	    //Send message when is new parcel
	    #sx_NewData := (#is_ObjectID <> #ss_Old_Object_ID) AND NOT (#is_ObjectID = '0');
	    // Save last value
	    #ss_Old_Object_ID := #is_ObjectID;

	END_REGION

	REGION 3 – Message array size validation

	    // Get size of the array.
	    #si_MaximumMessageLength := "FC_GetNrOfArrayEl"(#s_UDT_MessageArray.Bytes);

	    // Message array size validation.
	    #ss_Status.InvalidMessageArraySize := WORD_TO_INT(#ci_MessageLength) > #si_MaximumMessageLength;

	END_REGION


	REGION 4 – Message preparation

	    // FIFO full check.
	    IF NOT #iq_UDT_FifoHeader.Status.Full
	    THEN
	        // Errors and send pulse check.
	        IF NOT #ss_Status.FIFOError
	            AND NOT #ss_Status.InvalidMessageArraySize
	            AND #sx_NewData
	        THEN

	            REGION 4.1 – Header preparation

	                // Check sequence number. If it is equal or greater than 255 reset it to 1.
	                IF #iqdi_MessageSequenceNumber <= 255
	                THEN
	                    #iqdi_MessageSequenceNumber += 1;
	                ELSE
	                    #iqdi_MessageSequenceNumber := 1;
	                END_IF;

	                // Write parts of the header into structure.
	                #s_UDT_MessageHeader.SOM := #ci_Som;
	                #s_UDT_MessageHeader.SourceNode := INT_TO_BYTE(#ii_SourceNode);
	                #s_UDT_MessageHeader.DestinationNode := INT_TO_BYTE(#ii_DestinationNode);
	                #s_UDT_MessageHeader.SeqNumber := INT_TO_BYTE(#iqdi_MessageSequenceNumber);
	                #s_UDT_MessageHeader.DataLength := #ci_MessageLength;
	                #s_UDT_MessageHeader.NumMsg := 1;

	                //Convert string value to UDINT
	                #tudi_Temp := STRING_TO_UDINT(#is_ObjectID);

	                // Write parts of the body into structure.
	                #ss_MessageBody.MsgID := #ci_MsgID;
	                #ss_MessageBody.MsgLength := #ci_MsgLength;
	                #ss_MessageBody.ObjectID := UDINT_TO_DWORD(#tudi_Temp);
	                #ss_MessageBody.Eom := #ci_Eom;

	            END_REGION

	            REGION 4.2 – Convert message into array of bytes

	                // Initialize the header serialize position and convert header structure into array of bytes.
	                #sdi_SerializePosition := 0;
	                #si_SerializeStatus := Serialize(SRC_VARIABLE := #s_UDT_MessageHeader,
	                                                 DEST_ARRAY => #s_UDT_MessageArray.Bytes,
	                                                 POS := #sdi_SerializePosition);

	                // Initialize the body serialize position and convert header structure into array of bytes
	                #si_SerializeStatus := Serialize(SRC_VARIABLE := #ss_MessageBody,
	                                                 DEST_ARRAY => #s_UDT_MessageArray.Bytes,
	                                                 POS := #sdi_SerializePosition);

	            END_REGION

	            REGION 4.3 – Write message into the FIFO buffer

	                // Mode 'W' - Write FIFO record.
	                "FC_Fifo"(ic_Mode := 'W',
	                          qUDT_Status => #ss_Status.FIFOStatus,
	                          qx_Error => #ss_Status.FIFOError,
	                          qx_Warning => #ss_Status.FIFOWarning,
	                          iqv_Data := #s_UDT_MessageArray,
	                          iqUDT_FifoHeader := #iq_UDT_FifoHeader,
	                          iqv_DataBuffer := #iqs_FifoData);

	            END_REGION

	        END_IF;
	    ELSE
	        // If FIFO is full set FIFO main and FIFO full errors.
	        #ss_Status.FIFOError := TRUE;
	        #ss_Status.FIFOStatus.FifoFull := TRUE;
	    END_IF;

	END_REGION

	REGION 5 - Status

	    // Parametrization collective error output.
	    #qx_Error :=
	    #ss_Status.FIFOError
	    OR #ss_Status.InvalidTimeInterval
	    OR #ss_Status.InvalidMessageArraySize;

	    // Parametrization collective warning output.
	    #qx_Warning := #ss_Status.FIFOWarning;

	END_REGION
END_FUNCTION_BLOCK

FUNCTION_BLOCK "FB_MFC_Sort_SystemStatus"
{ S7_Optimized_Access := 'TRUE' }
VERSION : 0.1
// ATTRIBUTES
// AUTO_NUMBER = True
// BLOCK_NUMBER = 125
// END_ATTRIBUTES
   VAR_INPUT
      ii_SystemStatus { ExternalAccessible := 'False'; ExternalVisible := 'False'; ExternalWritable := 'False'} : Int;   // 1 - System stopped, 2 - System running
      iw_SystemMode { ExternalAccessible := 'False'; ExternalVisible := 'False'; ExternalWritable := 'False'} : Word;   // Bit value according to the documentation
      iui_LocationIdentifier { ExternalAccessible := 'False'; ExternalVisible := 'False'; ExternalWritable := 'False'} : UInt;   // Location Identifier
      ii_SourceNode { ExternalAccessible := 'False'; ExternalVisible := 'False'; ExternalWritable := 'False'} : Int;   // ID Source Node
      ii_DestinationNode { ExternalAccessible := 'False'; ExternalVisible := 'False'; ExternalWritable := 'False'} : Int;   // ID Destination Node
      ix_SendAllStatuses { ExternalAccessible := 'False'; ExternalVisible := 'False'; ExternalWritable := 'False'} : Bool;   // True - update all the statuses
   END_VAR

   VAR_OUTPUT
      qx_Error { ExternalAccessible := 'False'; ExternalVisible := 'False'; ExternalWritable := 'False'} : Bool;   // TRUE when collective block error occurred
      qx_Warning { ExternalAccessible := 'False'; ExternalVisible := 'False'; ExternalWritable := 'False'} : Bool;   // TRUE when collective block warning occurred
   END_VAR

   VAR_IN_OUT
      iq_UDT_FifoHeader : "UDT_FifoHeader";   // FIFO header
      iqs_FifoData : Array[*] of "UDT_MessageV2";   // FIFO data buffer
      iqdi_MessageSequenceNumber { ExternalAccessible := 'False'; ExternalVisible := 'False'; ExternalWritable := 'False'} : Int;   // Message number
   END_VAR

   VAR
      s_UDT_MessageArray { ExternalAccessible := 'False'; ExternalVisible := 'False'; ExternalWritable := 'False'; S7_SetPoint := 'False'} : "UDT_MessageV2";   // Message array byte
      s_UDT_MessageHeader { ExternalAccessible := 'False'; ExternalVisible := 'False'; ExternalWritable := 'False'; S7_SetPoint := 'False'} : "UDT_MFCSortMessageHeader";   // Message header
      s_F_TRIG_SendAllStatuses {InstructionName := 'F_TRIG'; LibVersion := '1.0'; ExternalAccessible := 'False'; ExternalVisible := 'False'; ExternalWritable := 'False'; S7_SetPoint := 'False'} : F_TRIG;   // Falling edge trigger from signal send all statuses
      ss_MessageBody { ExternalAccessible := 'False'; ExternalVisible := 'False'; ExternalWritable := 'False'} : Struct   // Message body
         MsgID { ExternalAccessible := 'False'; ExternalVisible := 'False'; ExternalWritable := 'False'} : Word;   // Message ID
         MsgLength { ExternalAccessible := 'False'; ExternalVisible := 'False'; ExternalWritable := 'False'} : Word;   // Message length
         LocationIdentifier { ExternalAccessible := 'False'; ExternalVisible := 'False'; ExternalWritable := 'False'} : Word;   // Location Identifier
         SystemStatus { ExternalAccessible := 'False'; ExternalVisible := 'False'; ExternalWritable := 'False'} : Byte;   // System status
         SystemMode { ExternalAccessible := 'False'; ExternalVisible := 'False'; ExternalWritable := 'False'} : Word;   // System mode
         Eom { ExternalAccessible := 'False'; ExternalVisible := 'False'; ExternalWritable := 'False'} : Byte;   // End of message
         Test { ExternalAccessible := 'False'; ExternalVisible := 'False'; ExternalWritable := 'False'} : Word := 16#0011;
         Test_1 { ExternalAccessible := 'False'; ExternalVisible := 'False'; ExternalWritable := 'False'} : Byte := 16#22;
      END_STRUCT;
      ss_Status { ExternalAccessible := 'False'; ExternalVisible := 'False'; ExternalWritable := 'False'} : Struct   // Status structure
         FIFOStatus { ExternalAccessible := 'False'; ExternalVisible := 'False'; ExternalWritable := 'False'} : "UDT_FifoStatus";
         FIFOError { ExternalAccessible := 'False'; ExternalVisible := 'False'; ExternalWritable := 'False'; S7_SetPoint := 'True'} : Bool;   //  FIFO error
         FIFOWarning { ExternalAccessible := 'False'; ExternalVisible := 'False'; ExternalWritable := 'False'; S7_SetPoint := 'True'} : Bool;   // FIFO warning
         InvalidMessageArraySize { ExternalAccessible := 'False'; ExternalVisible := 'False'; ExternalWritable := 'False'} : Bool;   // Message array is too short for message
         InvalidTimeInterval { ExternalAccessible := 'False'; ExternalVisible := 'False'; ExternalWritable := 'False'} : Bool;   // Heartbeat time interval lower than zero
      END_STRUCT;
      sw_SystemMode { ExternalAccessible := 'False'; ExternalVisible := 'False'; ExternalWritable := 'False'} : Word := 0;   // Bit value according to the documentation
      sw_Old_SystemMode { ExternalAccessible := 'False'; ExternalVisible := 'False'; ExternalWritable := 'False'} : Word;   // Data from previous PLC cycle: Maximum number of elements in message array
      sdi_SerializePosition { ExternalAccessible := 'False'; ExternalVisible := 'False'; ExternalWritable := 'False'} : DInt;   // Position in array where serialize finished writing data +1
      si_MaximumMessageLength { ExternalAccessible := 'False'; ExternalVisible := 'False'; ExternalWritable := 'False'} : Int;   // Maximum number of elements in message array
      si_SerializeStatus { ExternalAccessible := 'False'; ExternalVisible := 'False'; ExternalWritable := 'False'} : Int;   // Function serialize status
      si_SystemStatus { ExternalAccessible := 'False'; ExternalVisible := 'False'; ExternalWritable := 'False'} : Int := 0;   // 1 - System stopped, 2 - System running
      si_Old_SystemStatus { ExternalAccessible := 'False'; ExternalVisible := 'False'; ExternalWritable := 'False'} : Int := 0;   // Data from previous PLC cycle: 0 - System stopped, 1 - System running
      sx_NewData { ExternalAccessible := 'False'; ExternalVisible := 'False'; ExternalWritable := 'False'} : Bool;   // True - send a message to the MFC
   END_VAR

   VAR CONSTANT
      ci_MessageLength : Word := 16#0009;   // 10#0009 = 16#0009 - Message length
      ci_Som : Byte := 16#FD;   // Start of message
      ci_Eom : Byte := 16#FE;   // End of message
      ci_MsgID : Word := 16#00CC;   // 10#0204 = 16#00CC - Message ID
      ci_MsgLength : Word := 16#0005;   // 10#0005 = 16#0005 - Message length
   END_VAR


BEGIN
	(*
	----------------------------------------------------------------------------------------
	|                                                                                      |
	|  Copyright  2023             FORTNA Europe BV                                        |
	|  All Rights Reserved         Netherlands                                             |
	|                                                                                      |
	----------------------------------------------------------------------------------------
	Version history:
	Date        | Version   | Author       | Remark
	----------------------------------------------------------------------------------------
	21/07/2023  | 1.0       | S. Nikodem   | Release TIA 17 | DHL Munich 2023
	23/08/2023  | 1.1       | S. Theocharis| Serialise byte issue 0 - quick fix
	19/10/2023  | 1.2       | S. Nikodem   | Added "ix_SendAllStatuses" input and update for Serialize structure
	13/03/2023  | 1.3       | S. Nieswiec  | Updated for new Baseline
	02/05/2024  | 1.4       | J.Majer      | Datatype conversions changed from automatic to explicit, to accomodate IEC 61131-3 standard

	*)

	REGION 1 – FIFO header status update

	    // Mode 'S' - FIFO register status update.
	    "FC_Fifo"(ic_Mode := 'S',
	              qUDT_Status => #ss_Status.FIFOStatus,
	              qx_Error => #ss_Status.FIFOError,
	              qx_Warning => #ss_Status.FIFOWarning,
	              iqv_Data := #s_UDT_MessageArray,
	              iqUDT_FifoHeader := #iq_UDT_FifoHeader,
	              iqv_DataBuffer := #iqs_FifoData);

	END_REGION

	REGION 2 – Data preparation

	    // Prepare trigger
	    #s_F_TRIG_SendAllStatuses(CLK := #ix_SendAllStatuses);

	    // Data preparation
	    //  1 - System stopped, 2 - System running
	    #si_SystemStatus := #ii_SystemStatus;
	    // Bit value according to the documentation
	    #sw_SystemMode := #iw_SystemMode;

	    //Check if the data from the previous PLC cycle differs, if so, send a message to the MFC.
	    #sx_NewData := (#si_Old_SystemStatus <> #si_SystemStatus) OR (#sw_Old_SystemMode <> #sw_SystemMode) OR #s_F_TRIG_SendAllStatuses.Q;

	    // Copy data
	    #si_Old_SystemStatus := #si_SystemStatus;
	    #sw_Old_SystemMode := #sw_SystemMode;

	END_REGION

	REGION 3 – Message array size validation

	    // Get size of the array.
	    #si_MaximumMessageLength := "FC_GetNrOfArrayEl"(#s_UDT_MessageArray.Bytes);

	    // Message array size validation.
	    #ss_Status.InvalidMessageArraySize := WORD_TO_INT(#ci_MessageLength) > #si_MaximumMessageLength;

	END_REGION

	REGION 4 – Message preparation

	    // FIFO full check.
	    IF NOT #iq_UDT_FifoHeader.Status.Full
	    THEN
	        // Errors and send pulse check.
	        IF NOT #ss_Status.FIFOError
	            AND NOT #ss_Status.InvalidMessageArraySize
	            AND #sx_NewData
	        THEN

	            REGION 4.1 – Header preparation

	                // Check sequence number. If it is equal or greater than 255 reset it to 1.
	                IF #iqdi_MessageSequenceNumber <= 255
	                THEN
	                    #iqdi_MessageSequenceNumber += 1;
	                ELSE
	                    #iqdi_MessageSequenceNumber := 1;
	                END_IF;

	                // Write parts of the header into structure.
	                // Write parts of the header into structure.
	                #s_UDT_MessageHeader.SOM := #ci_Som;
	                #s_UDT_MessageHeader.SourceNode := INT_TO_BYTE(#ii_SourceNode);
	                #s_UDT_MessageHeader.DestinationNode := INT_TO_BYTE(#ii_DestinationNode);
	                #s_UDT_MessageHeader.SeqNumber := INT_TO_BYTE(#iqdi_MessageSequenceNumber);
	                #s_UDT_MessageHeader.DataLength := #ci_MessageLength;
	                #s_UDT_MessageHeader.NumMsg := 1;

	                // Write parts of the body into structure.
	                #ss_MessageBody.MsgID := #ci_MsgID;
	                #ss_MessageBody.MsgLength := #ci_MsgLength;
	                #ss_MessageBody.LocationIdentifier := DINT_TO_WORD(#iui_LocationIdentifier);
	                #ss_MessageBody.SystemStatus := INT_TO_BYTE(#si_SystemStatus);
	                #ss_MessageBody.SystemMode := #sw_SystemMode;
	                #ss_MessageBody.Eom := #ci_Eom;

	            END_REGION

	            REGION 4.2 – Convert message into array of bytes

	                // Initialize the header serialize position and convert header structure into array of bytes.
	                #sdi_SerializePosition := 0;
	                #si_SerializeStatus := Serialize(SRC_VARIABLE := #s_UDT_MessageHeader,
	                                                 DEST_ARRAY => #s_UDT_MessageArray.Bytes,
	                                                 POS := #sdi_SerializePosition);

	                #si_SerializeStatus := Serialize(SRC_VARIABLE := #ss_MessageBody.MsgID,
	                                                 DEST_ARRAY => #s_UDT_MessageArray.Bytes,
	                                                 POS := #sdi_SerializePosition);

	                #si_SerializeStatus := Serialize(SRC_VARIABLE := #ss_MessageBody.MsgLength,
	                                                 DEST_ARRAY => #s_UDT_MessageArray.Bytes,
	                                                 POS := #sdi_SerializePosition);

	                #si_SerializeStatus := Serialize(SRC_VARIABLE := #ss_MessageBody.LocationIdentifier,
	                                                 DEST_ARRAY => #s_UDT_MessageArray.Bytes,
	                                                 POS := #sdi_SerializePosition);

	                #si_SerializeStatus := Serialize(SRC_VARIABLE := #ss_MessageBody.SystemStatus,
	                                                 DEST_ARRAY => #s_UDT_MessageArray.Bytes,
	                                                 POS := #sdi_SerializePosition);

	                #si_SerializeStatus := Serialize(SRC_VARIABLE := #ss_MessageBody.SystemMode,
	                                                 DEST_ARRAY => #s_UDT_MessageArray.Bytes,
	                                                 POS := #sdi_SerializePosition);

	                #si_SerializeStatus := Serialize(SRC_VARIABLE := #ss_MessageBody.Eom,
	                                                 DEST_ARRAY => #s_UDT_MessageArray.Bytes,
	                                                 POS := #sdi_SerializePosition);

	            END_REGION

	            REGION 4.3 – Write message into the FIFO buffer

	                // Mode 'W' - Write FIFO record.
	                "FC_Fifo"(ic_Mode := 'W',
	                          qUDT_Status => #ss_Status.FIFOStatus,
	                          qx_Error => #ss_Status.FIFOError,
	                          qx_Warning => #ss_Status.FIFOWarning,
	                          iqv_Data := #s_UDT_MessageArray,
	                          iqUDT_FifoHeader := #iq_UDT_FifoHeader,
	                          iqv_DataBuffer := #iqs_FifoData);

	            END_REGION

	        END_IF;
	    ELSE
	        // If FIFO is full set FIFO main and FIFO full errors.
	        #ss_Status.FIFOError := TRUE;
	        #ss_Status.FIFOStatus.FifoFull := TRUE;
	    END_IF;

	END_REGION

	REGION 5 - Status

	    // Parametrization collective error output.
	    #qx_Error :=
	    #ss_Status.FIFOError
	    OR #ss_Status.InvalidTimeInterval
	    OR #ss_Status.InvalidMessageArraySize;

	    // Parametrization collective warning output.
	    #qx_Warning := #ss_Status.FIFOWarning;

	END_REGION
END_FUNCTION_BLOCK

FUNCTION_BLOCK "FB_MFC_Sort_TCPIPSend"
TITLE = FB_TCPIPSend
{ S7_Optimized_Access := 'TRUE' }
AUTHOR : MHSE
FAMILY : Communication
VERSION : 2.0
// ATTRIBUTES
// AUTO_NUMBER = True
// BLOCK_NUMBER = 127
// END_ATTRIBUTES
//Function block to send data from TCPIP.
   VAR_INPUT
      i_UDT_Connection { ExternalAccessible := 'False'; ExternalVisible := 'False'; ExternalWritable := 'False'} : "UDT_Connection";   // Connection parameters
      ix_EnableSend { ExternalAccessible := 'False'; ExternalVisible := 'False'; ExternalWritable := 'False'} : Bool;   // TRUE when send is enable
   END_VAR

   VAR_OUTPUT
      qx_Error { ExternalAccessible := 'False'; ExternalVisible := 'False'; ExternalWritable := 'False'} : Bool;   // TRUE when collective block error occurred
      qx_Warning { ExternalAccessible := 'False'; ExternalVisible := 'False'; ExternalWritable := 'False'} : Bool;   // TRUE when collective block warning occurred
   END_VAR

   VAR_IN_OUT
      iq_UDT_FifoLowHeader : "UDT_FifoHeader";   // Low priority FIFO header
      iqs_FifoLowData : Variant;   // Low priority FIFO data
      iq_UDT_FifoMediumHeader : "UDT_FifoHeader";   // Medium priority FIFO header
      iqs_FifoMediumData : Variant;   // Medium priority FIFO data
      iq_UDT_FifoHighHeader : "UDT_FifoHeader";   // High priority FIFO header
      iqs_FifoHighData : Variant;   // High priority FIFO data
   END_VAR

   VAR
      s_FB_TSEND {InstructionName := 'TSEND'; LibVersion := '4.0'; ExternalAccessible := 'False'; ExternalVisible := 'False'; ExternalWritable := 'False'; S7_SetPoint := 'False'} : TSEND;   // Siemens "TSEND" block - to send the data over TCPIP socket
      s_UDT_MessageArray { ExternalAccessible := 'False'; ExternalVisible := 'False'; ExternalWritable := 'False'; S7_SetPoint := 'False'} : "UDT_MessageV2";   // Message
      ss_TSEND { ExternalAccessible := 'False'; ExternalVisible := 'False'; ExternalWritable := 'False'} : Struct   // TSEND block structure
         Status { ExternalAccessible := 'False'; ExternalVisible := 'False'; ExternalWritable := 'False'} : Word;   //    TSEND - Status
         Request { ExternalAccessible := 'False'; ExternalVisible := 'False'; ExternalWritable := 'False'} : Bool;   //    TSEND - Request
         Busy { ExternalAccessible := 'False'; ExternalVisible := 'False'; ExternalWritable := 'False'} : Bool;   //    TSEND - Busy
         Done { ExternalAccessible := 'False'; ExternalVisible := 'False'; ExternalWritable := 'False'} : Bool;   //    TSEND - Done
         Error { ExternalAccessible := 'False'; ExternalVisible := 'False'; ExternalWritable := 'False'} : Bool;   //    TSEND - Error
      END_STRUCT;
      ss_Status { ExternalAccessible := 'False'; ExternalVisible := 'False'; ExternalWritable := 'False'} : Struct   // Status structure
         FIFOLowPriorityStatus { ExternalAccessible := 'False'; ExternalVisible := 'False'; ExternalWritable := 'False'} : "UDT_FifoStatus";
         FIFOMedPriorityStatus { ExternalAccessible := 'False'; ExternalVisible := 'False'; ExternalWritable := 'False'} : "UDT_FifoStatus";
         FIFOHighPriorityStatus { ExternalAccessible := 'False'; ExternalVisible := 'False'; ExternalWritable := 'False'} : "UDT_FifoStatus";
         FIFOLowPriorityError { ExternalAccessible := 'False'; ExternalVisible := 'False'; ExternalWritable := 'False'} : Bool;   // FIFO low priority error
         FIFOLowPriorityWarning { ExternalAccessible := 'False'; ExternalVisible := 'False'; ExternalWritable := 'False'} : Bool;   // FIFO low priority warning
         FIFOMedPriorityError { ExternalAccessible := 'False'; ExternalVisible := 'False'; ExternalWritable := 'False'} : Bool;   // FIFO medium priority error
         FIFOMedPriorityWarning { ExternalAccessible := 'False'; ExternalVisible := 'False'; ExternalWritable := 'False'} : Bool;   // FIFO medium priority warning
         FIFOHighPriorityError { ExternalAccessible := 'False'; ExternalVisible := 'False'; ExternalWritable := 'False'} : Bool;   // FIFO high priority error
         FIFOHighPriorityWarning { ExternalAccessible := 'False'; ExternalVisible := 'False'; ExternalWritable := 'False'} : Bool;   // FIFO high priority warning
         SendError { ExternalAccessible := 'False'; ExternalVisible := 'False'; ExternalWritable := 'False'} : Bool;   // Send operation error
      END_STRUCT;
      sw_BodyLength { ExternalAccessible := 'False'; ExternalVisible := 'False'; ExternalWritable := 'False'} : Word;   // Message body length
      sa_BodyLength { ExternalAccessible := 'False'; ExternalVisible := 'False'; ExternalWritable := 'False'} : Array[0..1] of Byte;
      si_MessageLength { ExternalAccessible := 'False'; ExternalVisible := 'False'; ExternalWritable := 'False'} : Int;   // Message length
      sx_MessageReady { ExternalAccessible := 'False'; ExternalVisible := 'False'; ExternalWritable := 'False'} : Bool;   // Message is ready to send
      sx_MessageRead { ExternalAccessible := 'False'; ExternalVisible := 'False'; ExternalWritable := 'False'} : Bool;   // Message has been read
      sx_MessageReadRequest { ExternalAccessible := 'False'; ExternalVisible := 'False'; ExternalWritable := 'False'} : Bool;   // Request to read message
      sx_FIFOError { ExternalAccessible := 'False'; ExternalVisible := 'False'; ExternalWritable := 'False'} : Bool;   // Summary FIFO error
      sdi_SerializePosition { ExternalAccessible := 'False'; ExternalVisible := 'False'; ExternalWritable := 'False'} : DInt;   // Position in array where serialize finished writing data +1
      si_SerializeStatus { ExternalAccessible := 'False'; ExternalVisible := 'False'; ExternalWritable := 'False'} : Int;   // Function serialize status
   END_VAR

   VAR CONSTANT
      ci_HeaderLength : Int := 8;   // Message header length
      ci_BodyLengthPosition : Int := 4;   // Position in header where message body length value starts
      cdi_POS : DInt := 2;
   END_VAR


BEGIN
	(*
	----------------------------------------------------------------------------------------
	|                                                                                      |
	|  Copyright  2023             FORTNA Europe BV                                        |
	|  All Rights Reserved         Netherlands                                             |
	|                                                                                      |
	----------------------------------------------------------------------------------------
	Version history:
	Date        | Version   | Author       | Remark
	----------------------------------------------------------------------------------------
	16/01/2023  | 1.0       | S. Nikodem   | Release TIA 17 | DHL Munich 2023
	13/03/2023  | 1.1       | S. Nieswiec  | Updated for new Baseline
	*)

	REGION 1 – Update FIFO header status bits

	    // Mode 'S' - High priority FIFO register status update.
	    "FC_Fifo"(ic_Mode := 'S',
	              qUDT_Status => #ss_Status.FIFOHighPriorityStatus,
	              qx_Error => #ss_Status.FIFOHighPriorityError,
	              qx_Warning => #ss_Status.FIFOHighPriorityWarning,
	              iqv_Data := #s_UDT_MessageArray,
	              iqUDT_FifoHeader := #iq_UDT_FifoHighHeader,
	              iqv_DataBuffer := #iqs_FifoHighData);

	    // Mode 'S' - Medium priority FIFO register status update.
	    "FC_Fifo"(ic_Mode := 'S',
	              qUDT_Status => #ss_Status.FIFOMedPriorityStatus,
	              qx_Error => #ss_Status.FIFOMedPriorityError,
	              qx_Warning => #ss_Status.FIFOMedPriorityWarning,
	              iqv_Data := #s_UDT_MessageArray,
	              iqUDT_FifoHeader := #iq_UDT_FifoMediumHeader,
	              iqv_DataBuffer := #iqs_FifoMediumData);

	    // Mode 'S' - Low priority FIFO register status update.
	    "FC_Fifo"(ic_Mode := 'S',
	              qUDT_Status => #ss_Status.FIFOLowPriorityStatus,
	              qx_Error => #ss_Status.FIFOLowPriorityError,
	              qx_Warning => #ss_Status.FIFOLowPriorityWarning,
	              iqv_Data := #s_UDT_MessageArray,
	              iqUDT_FifoHeader := #iq_UDT_FifoLowHeader,
	              iqv_DataBuffer := #iqs_FifoLowData);

	END_REGION

	REGION 2 – FIFO header summary error

	    #sx_FIFOError :=
	    #ss_Status.FIFOHighPriorityError
	    OR #ss_Status.FIFOMedPriorityError
	    OR #ss_Status.FIFOLowPriorityError;

	END_REGION

	REGION 3 – FIFO Read request

	    #sx_MessageReadRequest :=
	    #ix_EnableSend
	    AND NOT #sx_FIFOError
	    AND NOT #ss_TSEND.Error
	    AND #ss_TSEND.Status = 16#7000;

	END_REGION

	REGION 4 – Read the message from high priority FIFO data buffer

	    IF #sx_MessageReadRequest
	        AND NOT #iq_UDT_FifoHighHeader.Status.Empty
	        AND NOT #sx_MessageRead
	    THEN
	        // Mode 'R' - Read high priority FIFO record.
	        "FC_Fifo"(ic_Mode := 'R',
	                  qUDT_Status => #ss_Status.FIFOHighPriorityStatus,
	                  qx_Error => #ss_Status.FIFOHighPriorityError,
	                  qx_Warning => #ss_Status.FIFOHighPriorityWarning,
	                  iqv_Data := #s_UDT_MessageArray,
	                  iqUDT_FifoHeader := #iq_UDT_FifoHighHeader,
	                  iqv_DataBuffer := #iqs_FifoHighData);

	        #sx_MessageRead := TRUE;
	    END_IF;

	END_REGION

	REGION 5 – Read the message from medium priority FIFO data buffer

	    IF #sx_MessageReadRequest
	        AND #iq_UDT_FifoHighHeader.Status.Empty
	        AND NOT #iq_UDT_FifoMediumHeader.Status.Empty
	        AND NOT #sx_MessageRead
	    THEN
	        // Mode 'R' - Read medium priority FIFO record.
	        "FC_Fifo"(ic_Mode := 'R',
	                  qUDT_Status => #ss_Status.FIFOMedPriorityStatus,
	                  qx_Error => #ss_Status.FIFOMedPriorityError,
	                  qx_Warning => #ss_Status.FIFOMedPriorityWarning,
	                  iqv_Data := #s_UDT_MessageArray,
	                  iqUDT_FifoHeader := #iq_UDT_FifoMediumHeader,
	                  iqv_DataBuffer := #iqs_FifoMediumData);

	        #sx_MessageRead := TRUE;
	    END_IF;

	END_REGION

	REGION 6 – Read the message from low priority FIFO data buffer

	    IF #sx_MessageReadRequest
	        AND #iq_UDT_FifoHighHeader.Status.Empty
	        AND #iq_UDT_FifoMediumHeader.Status.Empty
	        AND NOT #iq_UDT_FifoLowHeader.Status.Empty
	        AND NOT #sx_MessageRead
	    THEN
	        #sx_MessageRead := TRUE;

	        // Mode 'R' - Read low priority FIFO record.
	        "FC_Fifo"(ic_Mode := 'R',
	                  qUDT_Status => #ss_Status.FIFOLowPriorityStatus,
	                  qx_Error => #ss_Status.FIFOLowPriorityError,
	                  qx_Warning => #ss_Status.FIFOLowPriorityWarning,
	                  iqv_Data := #s_UDT_MessageArray,
	                  iqUDT_FifoHeader := #iq_UDT_FifoLowHeader,
	                  iqv_DataBuffer := #iqs_FifoLowData);
	    END_IF;

	END_REGION

	REGION 7 – Message length

	    // Measuring the length of a read message.
	    IF #sx_MessageRead
	        AND NOT #sx_MessageReady
	    THEN
	        // Initialize the message length.
	        #si_MessageLength := 0;

	        // Get the length of the message by extracting the body length from the message header.
	        #sa_BodyLength[0] := #s_UDT_MessageArray.Bytes[#ci_BodyLengthPosition];
	        #sa_BodyLength[1] := #s_UDT_MessageArray.Bytes[#ci_BodyLengthPosition + 1];

	        #sdi_SerializePosition := 0;
	        #si_SerializeStatus := Deserialize(SRC_ARRAY := #sa_BodyLength,
	                                           DEST_VARIABLE => #sw_BodyLength,
	                                           POS := #sdi_SerializePosition);

	        #si_MessageLength := WORD_TO_INT(#sw_BodyLength) + #ci_HeaderLength + 1; // Add body, header and tail
	        #sx_MessageReady := TRUE;
	    END_IF;

	END_REGION

	REGION 8 – Send request

	    IF #sx_MessageRead
	        AND #sx_MessageReady
	    THEN
	        #ss_TSEND.Request := TRUE;
	    END_IF;

	END_REGION

	REGION 9 – Send data

	    #s_FB_TSEND(REQ := #ss_TSEND.Request,
	                ID := #i_UDT_Connection.ID,
	                LEN := INT_TO_UDINT(#si_MessageLength),
	                DONE => #ss_TSEND.Done,
	                BUSY => #ss_TSEND.Busy,
	                ERROR => #ss_TSEND.Error,
	                STATUS => #ss_TSEND.Status,
	                DATA := #s_UDT_MessageArray);

	    // Reset send request, message read and ready bits.
	    IF #ss_TSEND.Request
	        AND NOT #ss_TSEND.Busy
	        AND (#ss_TSEND.Done
	        OR #ss_TSEND.Status = 16#7000)
	    THEN
	        #ss_TSEND.Request := FALSE;
	        #sx_MessageRead := FALSE;
	        #sx_MessageReady := FALSE;
	    END_IF;

	    // Reset send error and TSEND status after correctly sent message.
	    IF #ss_TSEND.Done
	    THEN
	        #ss_Status.SendError := FALSE;
	    END_IF;

	    // Set send error and TSEND status if error occured.
	    IF #ss_TSEND.Error
	    THEN
	        #ss_Status.SendError := TRUE;
	    END_IF;

	END_REGION

	REGION 10 – Status

	    // Parametrization collective error output.
	    #qx_Error :=
	    #sx_FIFOError
	    OR #ss_Status.SendError;

	    // Parametrization collective warning output.
	    #qx_Warning :=
	    #ss_Status.FIFOHighPriorityWarning
	    OR #ss_Status.FIFOMedPriorityWarning
	    OR #ss_Status.FIFOLowPriorityWarning;

	END_REGION
END_FUNCTION_BLOCK

FUNCTION_BLOCK "FB_MFC_Sort_VIDResponse"
{ S7_Optimized_Access := 'TRUE' }
VERSION : 0.1
// ATTRIBUTES
// AUTO_NUMBER = True
// BLOCK_NUMBER = 128
// END_ATTRIBUTES
   VAR_INPUT
      ii_Object_ID { ExternalAccessible := 'False'; ExternalVisible := 'False'; ExternalWritable := 'False'} : Int;   // Parcel identifier
      i_ActualTimeDTL {InstructionName := 'DTL'; LibVersion := '1.0'; ExternalAccessible := 'False'; ExternalVisible := 'False'; ExternalWritable := 'False'} : DTL;   // Actual date and time in DTL
      ii_SourceNode { ExternalAccessible := 'False'; ExternalVisible := 'False'; ExternalWritable := 'False'} : Int;   // ID Source Node
      ii_DestinationNode { ExternalAccessible := 'False'; ExternalVisible := 'False'; ExternalWritable := 'False'} : Int;   // ID Destination Node
   END_VAR

   VAR_OUTPUT
      qx_Error { ExternalAccessible := 'False'; ExternalVisible := 'False'; ExternalWritable := 'False'} : Bool;   // TRUE when collective block error occurred
      qx_Warning { ExternalAccessible := 'False'; ExternalVisible := 'False'; ExternalWritable := 'False'} : Bool;   // TRUE when collective block warning occurred
   END_VAR

   VAR_IN_OUT
      iq_UDT_FifoHeader : "UDT_FifoHeader";   // FIFO header
      iqs_FifoData : Array[*] of "UDT_MessageV2";   // FIFO data buffer
      iqdi_MessageSequenceNumber { ExternalAccessible := 'False'; ExternalVisible := 'False'; ExternalWritable := 'False'} : Int;   // Message number
   END_VAR

   VAR
      s_UDT_MessageArray { ExternalAccessible := 'False'; ExternalVisible := 'False'; ExternalWritable := 'False'; S7_SetPoint := 'False'} : "UDT_MessageV2";   // Message array byte
      s_UDT_MessageHeader { ExternalAccessible := 'False'; ExternalVisible := 'False'; ExternalWritable := 'False'; S7_SetPoint := 'False'} : "UDT_MFCSortMessageHeader";   // Message header
      ss_MessageBody { ExternalAccessible := 'False'; ExternalVisible := 'False'; ExternalWritable := 'False'} : Struct   // Message body
         MsgID { ExternalAccessible := 'False'; ExternalVisible := 'False'; ExternalWritable := 'False'} : Word;   // Message ID
         MsgLength { ExternalAccessible := 'False'; ExternalVisible := 'False'; ExternalWritable := 'False'} : Word;   // Message length
         ObjectID { ExternalAccessible := 'False'; ExternalVisible := 'False'; ExternalWritable := 'False'} : Word;   // Parcel identifier
         VID { ExternalAccessible := 'False'; ExternalVisible := 'False'; ExternalWritable := 'False'} : Struct   // Virtual Item Identifier
            Year { ExternalAccessible := 'False'; ExternalVisible := 'False'; ExternalWritable := 'False'} : DWord;   // Year
            Month { ExternalAccessible := 'False'; ExternalVisible := 'False'; ExternalWritable := 'False'} : Word;   // Month
            Day { ExternalAccessible := 'False'; ExternalVisible := 'False'; ExternalWritable := 'False'} : Word;   // Day
            ObjectID { ExternalAccessible := 'False'; ExternalVisible := 'False'; ExternalWritable := 'False'} : Word;   // ObjectID
            Code1 { ExternalAccessible := 'False'; ExternalVisible := 'False'; ExternalWritable := 'False'} : Byte;   // Code1
            Code2 { ExternalAccessible := 'False'; ExternalVisible := 'False'; ExternalWritable := 'False'} : Byte;   // Code2
            Code3 { ExternalAccessible := 'False'; ExternalVisible := 'False'; ExternalWritable := 'False'} : Byte;   // Code3
            Code4 { ExternalAccessible := 'False'; ExternalVisible := 'False'; ExternalWritable := 'False'} : Byte;   // Code4
            Code5 { ExternalAccessible := 'False'; ExternalVisible := 'False'; ExternalWritable := 'False'} : Byte;   // Code5
            Code6 { ExternalAccessible := 'False'; ExternalVisible := 'False'; ExternalWritable := 'False'} : Byte;   // Code6
         END_STRUCT;
         Eom { ExternalAccessible := 'False'; ExternalVisible := 'False'; ExternalWritable := 'False'} : Byte;   // End of message
      END_STRUCT;
      ss_Status { ExternalAccessible := 'False'; ExternalVisible := 'False'; ExternalWritable := 'False'} : Struct   // Status structure
         FIFOStatus { ExternalAccessible := 'False'; ExternalVisible := 'False'; ExternalWritable := 'False'} : "UDT_FifoStatus";
         FIFOError { ExternalAccessible := 'False'; ExternalVisible := 'False'; ExternalWritable := 'False'; S7_SetPoint := 'True'} : Bool;   //  FIFO error
         FIFOWarning { ExternalAccessible := 'False'; ExternalVisible := 'False'; ExternalWritable := 'False'; S7_SetPoint := 'True'} : Bool;   // FIFO warning
         InvalidMessageArraySize { ExternalAccessible := 'False'; ExternalVisible := 'False'; ExternalWritable := 'False'} : Bool;   // Message array is too short for message
         InvalidTimeInterval { ExternalAccessible := 'False'; ExternalVisible := 'False'; ExternalWritable := 'False'} : Bool;   // Heartbeat time interval lower than zero
      END_STRUCT;
      sdi_SerializePosition { ExternalAccessible := 'False'; ExternalVisible := 'False'; ExternalWritable := 'False'} : DInt;   // Position in array where serialize finished writing data +1
      si_MaximumMessageLength { ExternalAccessible := 'False'; ExternalVisible := 'False'; ExternalWritable := 'False'} : Int;   // Maximum number of elements in message array
      si_SerializeStatus { ExternalAccessible := 'False'; ExternalVisible := 'False'; ExternalWritable := 'False'} : Int;   // Function serialize status
      ss_VID { ExternalAccessible := 'False'; ExternalVisible := 'False'; ExternalWritable := 'False'} : Struct   // Virtual Item Identifier
         Year { ExternalAccessible := 'False'; ExternalVisible := 'False'; ExternalWritable := 'False'} : DWord;   // Year
         Month { ExternalAccessible := 'False'; ExternalVisible := 'False'; ExternalWritable := 'False'} : Word;   // Month
         Day { ExternalAccessible := 'False'; ExternalVisible := 'False'; ExternalWritable := 'False'} : Word;   // Day
         ObjectID { ExternalAccessible := 'False'; ExternalVisible := 'False'; ExternalWritable := 'False'} : Word;   // ObjectID
         Code1 { ExternalAccessible := 'False'; ExternalVisible := 'False'; ExternalWritable := 'False'} : Byte;   // Code1
         Code2 { ExternalAccessible := 'False'; ExternalVisible := 'False'; ExternalWritable := 'False'} : Byte;   // Code2
         Code3 { ExternalAccessible := 'False'; ExternalVisible := 'False'; ExternalWritable := 'False'} : Byte;   // Code3
         Code4 { ExternalAccessible := 'False'; ExternalVisible := 'False'; ExternalWritable := 'False'} : Byte;   // Code4
         Code5 { ExternalAccessible := 'False'; ExternalVisible := 'False'; ExternalWritable := 'False'} : Byte;   // Code5
         Code6 { ExternalAccessible := 'False'; ExternalVisible := 'False'; ExternalWritable := 'False'} : Byte;   // Code6
      END_STRUCT;
      si_Old_Object_ID { ExternalAccessible := 'False'; ExternalVisible := 'False'; ExternalWritable := 'False'} : Int;   // Value from previous PLC cycle
      sx_NewData { ExternalAccessible := 'False'; ExternalVisible := 'False'; ExternalWritable := 'False'} : Bool;   // True - send a message to the MFC
   END_VAR

   VAR CONSTANT
      ci_MessageLength : Word := 16#0016;   // 10#0021 = 16#0016 - Message length
      ci_Som : Byte := 16#FD;   // Start of message
      ci_Eom : Byte := 16#FE;   // End of message
      ci_MsgID : Word := 16#00C9;   // 10#0201 = 16#00C9 - Message ID
      ci_MsgLength : Word := 16#0011;   // 10#0017 = 16#0011 - Message length
   END_VAR


BEGIN
	(*
	----------------------------------------------------------------------------------------
	|                                                                                      |
	|  Copyright  2023             FORTNA Europe BV                                        |
	|  All Rights Reserved         Netherlands                                             |
	|                                                                                      |
	----------------------------------------------------------------------------------------
	Version history:
	Date        | Version   | Author       | Remark
	----------------------------------------------------------------------------------------
	05/01/2023  | 1.0       | S. Nikodem   | Release TIA 17 | DHL Munich 2023
	13/03/2023  | 1.1       | S. Nieswiec  | Updated for new Baseline
	02/05/2024  | 1.2       | J.Majer      | Datatype conversions changed from automatic to explicit, to accomodate IEC 61131-3 standard

	*)

	REGION 1 – FIFO header status update

	    // Mode 'S' - FIFO register status update.
	    "FC_Fifo"(ic_Mode := 'S',
	              qUDT_Status => #ss_Status.FIFOStatus,
	              qx_Error => #ss_Status.FIFOError,
	              qx_Warning => #ss_Status.FIFOWarning,
	              iqv_Data := #s_UDT_MessageArray,
	              iqUDT_FifoHeader := #iq_UDT_FifoHeader,
	              iqv_DataBuffer := #iqs_FifoData);

	END_REGION

	REGION 2 – Data preparation

	    #ss_MessageBody.VID.Year := UINT_TO_DWORD(#i_ActualTimeDTL.YEAR);
	    #ss_MessageBody.VID.Month := UINT_TO_WORD(#i_ActualTimeDTL.MONTH);
	    #ss_MessageBody.VID.Day := UINT_TO_WORD(#i_ActualTimeDTL.DAY);
	    #ss_MessageBody.VID.ObjectID := INT_TO_WORD(#ii_Object_ID);
	    #ss_MessageBody.VID.Code1 := 0;
	    #ss_MessageBody.VID.Code2 := 0;
	    #ss_MessageBody.VID.Code3 := 0;
	    #ss_MessageBody.VID.Code4 := 0;
	    #ss_MessageBody.VID.Code5 := 0;
	    #ss_MessageBody.VID.Code6 := 0;


	    //Send message when is new parcel
	    #sx_NewData := (#ii_Object_ID <> #si_Old_Object_ID) AND (#ii_Object_ID <> 0);
	    // Save last value
	    #si_Old_Object_ID := #ii_Object_ID;


	END_REGION

	REGION 3 – Message array size validation

	    // Get size of the array.
	    #si_MaximumMessageLength := "FC_GetNrOfArrayEl"(#s_UDT_MessageArray.Bytes);

	    // Message array size validation.
	    #ss_Status.InvalidMessageArraySize := WORD_TO_INT(#ci_MessageLength) > #si_MaximumMessageLength;

	END_REGION


	REGION 4 – Message preparation

	    // FIFO full check.
	    IF NOT #iq_UDT_FifoHeader.Status.Full
	    THEN
	        // Errors and send pulse check.
	        IF NOT #ss_Status.FIFOError
	            AND NOT #ss_Status.InvalidMessageArraySize
	            AND #sx_NewData
	        THEN

	            REGION 4.1 – Header preparation

	                // Check sequence number. If it is equal or greater than 255 reset it to 1.
	                IF #iqdi_MessageSequenceNumber <= 255
	                THEN
	                    #iqdi_MessageSequenceNumber += 1;
	                ELSE
	                    #iqdi_MessageSequenceNumber := 1;
	                END_IF;


	                // Write parts of the header into structure.
	                #s_UDT_MessageHeader.SOM := #ci_Som;
	                #s_UDT_MessageHeader.SourceNode := INT_TO_BYTE(#ii_SourceNode);
	                #s_UDT_MessageHeader.DestinationNode := INT_TO_BYTE(#ii_DestinationNode);
	                #s_UDT_MessageHeader.SeqNumber := INT_TO_BYTE(#iqdi_MessageSequenceNumber);
	                #s_UDT_MessageHeader.DataLength := #ci_MessageLength;
	                #s_UDT_MessageHeader.NumMsg := 1;

	                // Write parts of the body into structure.
	                #ss_MessageBody.MsgID := #ci_MsgID;
	                #ss_MessageBody.MsgLength := #ci_MsgLength;
	                #ss_MessageBody.ObjectID := INT_TO_WORD(#ii_Object_ID);
	                #ss_MessageBody.VID := #ss_VID;
	                #ss_MessageBody.Eom := #ci_Eom;

	            END_REGION

	            REGION 4.2 – Convert message into array of bytes

	                // Initialize the header serialize position and convert header structure into array of bytes.
	                #sdi_SerializePosition := 0;
	                #si_SerializeStatus := Serialize(SRC_VARIABLE := #s_UDT_MessageHeader,
	                                                 DEST_ARRAY => #s_UDT_MessageArray.Bytes,
	                                                 POS := #sdi_SerializePosition);

	                // Initialize the body serialize position and convert header structure into array of bytes
	                #si_SerializeStatus := Serialize(SRC_VARIABLE := #ss_MessageBody,
	                                                 DEST_ARRAY => #s_UDT_MessageArray.Bytes,
	                                                 POS := #sdi_SerializePosition);

	            END_REGION

	            REGION 4.3 – Write message into the FIFO buffer

	                // Mode 'W' - Write FIFO record.
	                "FC_Fifo"(ic_Mode := 'W',
	                          qUDT_Status => #ss_Status.FIFOStatus,
	                          qx_Error => #ss_Status.FIFOError,
	                          qx_Warning => #ss_Status.FIFOWarning,
	                          iqv_Data := #s_UDT_MessageArray,
	                          iqUDT_FifoHeader := #iq_UDT_FifoHeader,
	                          iqv_DataBuffer := #iqs_FifoData);

	            END_REGION

	        END_IF;
	    ELSE
	        // If FIFO is full set FIFO main and FIFO full errors.
	        #ss_Status.FIFOError := TRUE;
	        #ss_Status.FIFOStatus.FifoFull := TRUE;
	    END_IF;

	END_REGION

	REGION 5 - Status

	    // Parametrization collective error output.
	    #qx_Error :=
	    #ss_Status.FIFOError
	    OR #ss_Status.InvalidTimeInterval
	    OR #ss_Status.InvalidMessageArraySize;

	    // Parametrization collective warning output.
	    #qx_Warning := #ss_Status.FIFOWarning;

	END_REGION
END_FUNCTION_BLOCK

FUNCTION_BLOCK "FB_MFC_Sort_VIDResponse_ASCII"
{ S7_Optimized_Access := 'TRUE' }
VERSION : 0.1
// ATTRIBUTES
// AUTO_NUMBER = True
// BLOCK_NUMBER = 129
// END_ATTRIBUTES
   VAR_INPUT
      is_ObjectID { ExternalAccessible := 'False'; ExternalVisible := 'False'; ExternalWritable := 'False'} : String[10];   // Parcel identifier
      ii_SorterID { ExternalAccessible := 'False'; ExternalVisible := 'False'; ExternalWritable := 'False'} : Int;   // Sorter identifier
      i_ActualTimeDTL {InstructionName := 'DTL'; LibVersion := '1.0'; ExternalAccessible := 'False'; ExternalVisible := 'False'; ExternalWritable := 'False'} : DTL;   // Actual date and time in DTL
   END_VAR

   VAR_OUTPUT
      qx_Error { ExternalAccessible := 'False'; ExternalVisible := 'False'; ExternalWritable := 'False'} : Bool;   // TRUE when collective block error occurred
      qx_Warning { ExternalAccessible := 'False'; ExternalVisible := 'False'; ExternalWritable := 'False'} : Bool;   // TRUE when collective block warning occurred
   END_VAR

   VAR_IN_OUT
      iq_UDT_FifoHeader : "UDT_FifoHeader";   // FIFO header
      iqs_FifoData : Array[*] of "UDT_MessageV2";   // FIFO data buffer
      iqdi_MessageSequenceNumber { ExternalAccessible := 'False'; ExternalVisible := 'False'; ExternalWritable := 'False'} : Int;   // Message number
   END_VAR

   VAR
      s_UDT_MessageArray { ExternalAccessible := 'False'; ExternalVisible := 'False'; ExternalWritable := 'False'; S7_SetPoint := 'False'} : "UDT_MessageV2";   // Message array byte
      s_UDT_MessageHeader { ExternalAccessible := 'False'; ExternalVisible := 'False'; ExternalWritable := 'False'; S7_SetPoint := 'False'} : "UDT_MFCSortMessageHeader";   // Message header
      ss_MessageBody { ExternalAccessible := 'False'; ExternalVisible := 'False'; ExternalWritable := 'False'} : Struct   // Message body
         MsgID { ExternalAccessible := 'False'; ExternalVisible := 'False'; ExternalWritable := 'False'} : Word;   // Message ID
         MsgLength { ExternalAccessible := 'False'; ExternalVisible := 'False'; ExternalWritable := 'False'} : Word;   // Message length
         ObjectID { ExternalAccessible := 'False'; ExternalVisible := 'False'; ExternalWritable := 'False'} : String[10];   // Parcel identifier
         VID { ExternalAccessible := 'False'; ExternalVisible := 'False'; ExternalWritable := 'False'} : Array[0..15] of Byte;   // Virtual Item Identifier
         Eom { ExternalAccessible := 'False'; ExternalVisible := 'False'; ExternalWritable := 'False'} : Byte;   // End of message
      END_STRUCT;
      ss_Status { ExternalAccessible := 'False'; ExternalVisible := 'False'; ExternalWritable := 'False'} : Struct   // Status structure
         FIFOStatus { ExternalAccessible := 'False'; ExternalVisible := 'False'; ExternalWritable := 'False'} : "UDT_FifoStatus";
         HTAReturn { ExternalAccessible := 'False'; ExternalVisible := 'False'; ExternalWritable := 'False'} : Struct   // Status structure from HTA function
            Month { ExternalAccessible := 'False'; ExternalVisible := 'False'; ExternalWritable := 'False'} : Word;   // HTA_Month
            Day { ExternalAccessible := 'False'; ExternalVisible := 'False'; ExternalWritable := 'False'} : Word;   // HTA_Day
         END_STRUCT;
         FIFOError { ExternalAccessible := 'False'; ExternalVisible := 'False'; ExternalWritable := 'False'; S7_SetPoint := 'True'} : Bool;   //  FIFO error
         FIFOWarning { ExternalAccessible := 'False'; ExternalVisible := 'False'; ExternalWritable := 'False'; S7_SetPoint := 'True'} : Bool;   // FIFO warning
         InvalidMessageArraySize { ExternalAccessible := 'False'; ExternalVisible := 'False'; ExternalWritable := 'False'} : Bool;   // Message array is too short for message
         InvalidTimeInterval { ExternalAccessible := 'False'; ExternalVisible := 'False'; ExternalWritable := 'False'} : Bool;   // Heartbeat time interval lower than zero
         InvalidInputData { ExternalAccessible := 'False'; ExternalVisible := 'False'; ExternalWritable := 'False'} : Bool;   // Input is not in range
      END_STRUCT;
      ss_VID { ExternalAccessible := 'False'; ExternalVisible := 'False'; ExternalWritable := 'False'} : String;   // Virtual Item Identifier
      sa_VIDBytes { ExternalAccessible := 'False'; ExternalVisible := 'False'; ExternalWritable := 'False'} : Array[1..16] of Byte;   // VID  - array with data in ASCII
      sdi_SerializePosition { ExternalAccessible := 'False'; ExternalVisible := 'False'; ExternalWritable := 'False'} : DInt;   // Position in array where serialize finished writing data +1
      sdi_VIDCode { ExternalAccessible := 'False'; ExternalVisible := 'False'; ExternalWritable := 'False'} : DInt;   // VID Code
      si_MaximumMessageLength { ExternalAccessible := 'False'; ExternalVisible := 'False'; ExternalWritable := 'False'} : Int;   // Maximum number of elements in message array
      si_SerializeStatus { ExternalAccessible := 'False'; ExternalVisible := 'False'; ExternalWritable := 'False'} : Int;   // Function serialize status
      ss_OldObjectID { ExternalAccessible := 'False'; ExternalVisible := 'False'; ExternalWritable := 'False'} : String[10];   // Value from previous PLC cycle
      sx_NewData { ExternalAccessible := 'False'; ExternalVisible := 'False'; ExternalWritable := 'False'} : Bool;   // True - prepare data and send a message to the MFC
   END_VAR

   VAR_TEMP
      ts_StringDate : Struct   // Temporary memory with string value
         Year : String;
         Month : String;
         Day : String;
         SorterID : String;
         Code : String;
      END_STRUCT;
      ti_Loop : Int;   // Loop counter
      ti_ObjectID : UDInt;   // Parcel identifier
   END_VAR

   VAR CONSTANT
      ci_MessageLength : Word := 16#0016;   // 10#0021 = 16#0016 - Message length
      ci_Som : Byte := 16#FD;   // Start of message
      ci_Eom : Byte := 16#FE;   // End of message
      ci_MsgID : Word := 16#00C9;   // 10#0201 = 16#00C9 - Message ID
      ci_MsgLength : Word := 16#0012;   // 10#0018 = 16#0012 - Message length
      ci_SourceNode : Int := 1;   // 1 - PLC ID Source Node
      ci_DestinationNode : Int := 2;   // 2 - MFC ID Destination Node
   END_VAR


BEGIN
	(*
	----------------------------------------------------------------------------------------
	|                                                                                      |
	|  Copyright  2023             FORTNA Europe BV                                        |
	|  All Rights Reserved         Netherlands                                             |
	|                                                                                      |
	----------------------------------------------------------------------------------------
	Version history:
	Date        | Version   | Author       | Remark
	----------------------------------------------------------------------------------------
	27/04/2023  | 1.0       | S. Nikodem   | Release TIA 17 | DHL Munich 2023
	13/03/2023  | 1.1       | S. Nieswiec  | Updated for new Baseline
	02/05/2024  | 1.2       | J.Majer      | Datatype conversions changed from automatic to explicit, to accomodate IEC 61131-3 standard

	*)

	REGION 1 – FIFO header status update

	    // Mode 'S' - FIFO register status update.
	    "FC_Fifo"(ic_Mode := 'S',
	              qUDT_Status => #ss_Status.FIFOStatus,
	              qx_Error => #ss_Status.FIFOError,
	              qx_Warning => #ss_Status.FIFOWarning,
	              iqv_Data := #s_UDT_MessageArray,
	              iqUDT_FifoHeader := #iq_UDT_FifoHeader,
	              iqv_DataBuffer := #iqs_FifoData);

	END_REGION

	REGION 2 - Check input data if are if range

	    //Convert 'is_ObjectID' to numeric variable
	    #ti_ObjectID := STRING_TO_UDINT(#is_ObjectID);

	    IF (#ti_ObjectID < 0)
	        OR (#ii_SorterID < 0)
	        OR (#ii_SorterID > 99)
	    THEN
	        #ss_Status.InvalidInputData := True;
	    ELSE
	        #ss_Status.InvalidInputData := FALSE;
	    END_IF;

	END_REGION

	REGION 3 – Data preparation

	    //Send message when is new parcel
	    #sx_NewData := (#is_ObjectID <> #ss_OldObjectID) AND NOT (#is_ObjectID = '0');
	    // Save last value
	    #ss_OldObjectID := #is_ObjectID;

	END_REGION

	REGION 4 – Message array size validation

	    // Get size of the array.
	    #si_MaximumMessageLength := "FC_GetNrOfArrayEl"(#s_UDT_MessageArray.Bytes);

	    // Message array size validation.
	    #ss_Status.InvalidMessageArraySize := WORD_TO_INT(#ci_MessageLength) > #si_MaximumMessageLength;

	END_REGION

	REGION 5 – Message preparation

	    // FIFO full check.
	    IF NOT #iq_UDT_FifoHeader.Status.Full
	    THEN
	        // Errors and send pulse check.
	        IF NOT #ss_Status.FIFOError
	            AND NOT #ss_Status.InvalidMessageArraySize
	            AND NOT #ss_Status.InvalidInputData
	            AND #sx_NewData
	        THEN

	            REGION 5.1 – VID preparation

	                // Convert the year into a character string
	                VAL_STRG(IN := #i_ActualTimeDTL.YEAR,
	                         SIZE := 4,
	                         PREC := 0,
	                         FORMAT := 0,
	                         P := 1,
	                         OUT => #ts_StringDate.Year);

	                // Using the HTA function, convert date into a string format
	                #ss_Status.HTAReturn.Month := HTA(IN := WORD_TO_BYTE(INT_TO_BCD16((USINT_TO_INT(#i_ActualTimeDTL.MONTH)))), N := 1, OUT => #ts_StringDate.Month);   // Convert the month
	                #ss_Status.HTAReturn.Day := HTA(IN := WORD_TO_BYTE(INT_TO_BCD16((USINT_TO_INT(#i_ActualTimeDTL.DAY)))), N := 1, OUT => #ts_StringDate.Day);         // Convert the day

	                //Convert Sorter ID value from number to string
	                #ts_StringDate.SorterID := INT_TO_STRING(#ii_SorterID);

	                //Delete sing '+' from string value
	                IF #ts_StringDate.SorterID[1] = '+' THEN
	                    #ts_StringDate.SorterID := DELETE(IN := #ts_StringDate.SorterID, L := 1, P := 1);
	                END_IF;

	                //Add zero when the variable size is to small
	                IF #ii_SorterID < 10 THEN
	                    #ts_StringDate.SorterID := INSERT(IN1 := #ts_StringDate.SorterID, IN2 := '0', P := 0);
	                END_IF;

	                //Creat ID code - value 000 001 to 999 999
	                #sdi_VIDCode += 1;

	                IF #sdi_VIDCode > 999999 THEN
	                    #sdi_VIDCode := 0;
	                END_IF;

	                //Convert VID code value from number to string
	                #ts_StringDate.Code := DINT_TO_STRING(#sdi_VIDCode);

	                //Delete sing '+' from string
	                IF #ts_StringDate.Code[1] = '+' THEN
	                    #ts_StringDate.Code := DELETE(IN := #ts_StringDate.Code, L := 1, P := 1);
	                END_IF;

	                //Add zero when the variable size is to small
	                IF #sdi_VIDCode < 10 THEN
	                    #ts_StringDate.Code := INSERT(IN1 := #ts_StringDate.Code, IN2 := '00000', P := 0);
	                ELSIF #sdi_VIDCode < 100 THEN
	                    #ts_StringDate.Code := INSERT(IN1 := #ts_StringDate.Code, IN2 := '0000', P := 0);
	                ELSIF #sdi_VIDCode < 1000 THEN
	                    #ts_StringDate.Code := INSERT(IN1 := #ts_StringDate.Code, IN2 := '000', P := 0);
	                ELSIF #sdi_VIDCode < 10000 THEN
	                    #ts_StringDate.Code := INSERT(IN1 := #ts_StringDate.Code, IN2 := '00', P := 0);
	                ELSIF #sdi_VIDCode < 100000 THEN
	                    #ts_StringDate.Code := INSERT(IN1 := #ts_StringDate.Code, IN2 := '0', P := 0);
	                END_IF;

	                //Combine strings
	                #ss_VID := (CONCAT(IN1 := #ts_StringDate.Year,
	                                   IN2 := #ts_StringDate.Month,
	                                   IN3 := #ts_StringDate.Day,
	                                   IN4 := #ts_StringDate.SorterID,
	                                   IN5 := #ts_StringDate.Code));

	                //Convert string value to ASCII
	                FOR #ti_Loop := 1 TO 16 DO
	                    #sa_VIDBytes[#ti_Loop] := CHAR_TO_BYTE(#ss_VID[#ti_Loop]);
	                END_FOR;

	            END_REGION

	            REGION 5.2 – Header preparation

	                // Check sequence number. If it is equal or greater than 255 reset it to 1.
	                IF #iqdi_MessageSequenceNumber <= 255
	                THEN
	                    #iqdi_MessageSequenceNumber += 1;
	                ELSE
	                    #iqdi_MessageSequenceNumber := 1;
	                END_IF;

	                // Write parts of the header into structure.
	                #s_UDT_MessageHeader.SOM := #ci_Som;
	                #s_UDT_MessageHeader.SourceNode := INT_TO_BYTE(#ci_SourceNode);
	                #s_UDT_MessageHeader.DestinationNode := INT_TO_BYTE(#ci_DestinationNode);
	                #s_UDT_MessageHeader.SeqNumber := INT_TO_BYTE(#iqdi_MessageSequenceNumber);
	                #s_UDT_MessageHeader.DataLength := #ci_MessageLength;
	                #s_UDT_MessageHeader.NumMsg := 1;

	                // Write parts of the body into structure.
	                #ss_MessageBody.MsgID := #ci_MsgID;
	                #ss_MessageBody.MsgLength := #ci_MsgLength;
	                #ss_MessageBody.ObjectID := #is_ObjectID;
	                #ss_MessageBody.VID := #sa_VIDBytes;
	                #ss_MessageBody.Eom := #ci_Eom;

	            END_REGION

	            REGION 5.3 – Convert message into array of bytes

	                // Initialize the header serialize position and convert header structure into array of bytes.
	                #sdi_SerializePosition := 0;
	                #si_SerializeStatus := Serialize(SRC_VARIABLE := #s_UDT_MessageHeader,
	                                                 DEST_ARRAY => #s_UDT_MessageArray.Bytes,
	                                                 POS := #sdi_SerializePosition);

	                // Initialize the body serialize position and convert header structure into array of bytes
	                #si_SerializeStatus := Serialize(SRC_VARIABLE := #ss_MessageBody,
	                                                 DEST_ARRAY => #s_UDT_MessageArray.Bytes,
	                                                 POS := #sdi_SerializePosition);

	            END_REGION

	            REGION 5.4 – Write message into the FIFO buffer

	                // Mode 'W' - Write FIFO record.
	                "FC_Fifo"(ic_Mode := 'W',
	                          qUDT_Status => #ss_Status.FIFOStatus,
	                          qx_Error => #ss_Status.FIFOError,
	                          qx_Warning => #ss_Status.FIFOWarning,
	                          iqv_Data := #s_UDT_MessageArray,
	                          iqUDT_FifoHeader := #iq_UDT_FifoHeader,
	                          iqv_DataBuffer := #iqs_FifoData);

	            END_REGION

	        END_IF;
	    ELSE
	        // If FIFO is full set FIFO main and FIFO full errors.
	        #ss_Status.FIFOError := TRUE;
	        #ss_Status.FIFOStatus.FifoFull := TRUE;
	    END_IF;

	END_REGION

	REGION 6 - Status

	    // Parametrization collective error output.
	    #qx_Error :=
	    #ss_Status.FIFOError
	    OR #ss_Status.InvalidTimeInterval
	    OR #ss_Status.InvalidMessageArraySize
	    OR #ss_Status.InvalidInputData;

	    // Parametrization collective warning output.
	    #qx_Warning := #ss_Status.FIFOWarning;

	END_REGION
END_FUNCTION_BLOCK

FUNCTION_BLOCK "FB_MFC_Sort_Destination"
{ S7_Optimized_Access := 'TRUE' }
VERSION : 0.1
// ATTRIBUTES
// AUTO_NUMBER = True
// BLOCK_NUMBER = 248
// END_ATTRIBUTES
   VAR_INPUT
      ii_GINRangeStart { ExternalAccessible := 'False'; ExternalVisible := 'False'; ExternalWritable := 'False'} : Int := 1;   // GIN range start value
      ii_GINRangeEnd { ExternalAccessible := 'False'; ExternalVisible := 'False'; ExternalWritable := 'False'} : Int := 100;   // GIN range end value
      ii_SourceNode { ExternalAccessible := 'False'; ExternalVisible := 'False'; ExternalWritable := 'False'} : Int;   // Source Node
      ii_DestinationNode { ExternalAccessible := 'False'; ExternalVisible := 'False'; ExternalWritable := 'False'} : Int;   // Destination Node
   END_VAR

   VAR_IN_OUT
      iqdi_MessageSequenceNumber { ExternalAccessible := 'False'; ExternalVisible := 'False'; ExternalWritable := 'False'} : Int;   // Message number
      iq_UDT_FifoHeader : "UDT_FifoHeader";   // FIFO header
      iqs_FifoData : Array[*] of "UDT_MessageV2";   // FIFO data buffer
      iq_UDT_MFCParcelDestination : "UDT_MFCParcelDestination";   // Structure received from MFC with destination commands for the package (ObjectID)
   END_VAR

   VAR
      FB_MFC_Sort_SortResult_Instance { ExternalAccessible := 'False'; ExternalVisible := 'False'; ExternalWritable := 'False'; S7_SetPoint := 'False'} : "FB_MFC_Sort_SortResult";
      sx_NewDataGinNumber { ExternalAccessible := 'False'; ExternalVisible := 'False'; ExternalWritable := 'False'} : Int;
      ss_Counter { ExternalAccessible := 'False'; ExternalVisible := 'False'; ExternalWritable := 'False'} : Struct   // Counters for statistics
         NewData { ExternalAccessible := 'False'; ExternalVisible := 'False'; ExternalWritable := 'False'} : UDInt;
         CombinedData { ExternalAccessible := 'False'; ExternalVisible := 'False'; ExternalWritable := 'False'} : UDInt;
         DataNotMerged { ExternalAccessible := 'False'; ExternalVisible := 'False'; ExternalWritable := 'False'} : UDInt;
         DestinationResent { ExternalAccessible := 'False'; ExternalVisible := 'False'; ExternalWritable := 'False'} : UDInt;
         LateDestination { ExternalAccessible := 'False'; ExternalVisible := 'False'; ExternalWritable := 'False'} : UDInt;
      END_STRUCT;
   END_VAR

   VAR_TEMP
      ti_GINLoop : Int;
      ti_DestinationLoop : Int;
   END_VAR


BEGIN
	(*
	----------------------------------------------------------------------------------------
	|                                                                                      |
	|  Copyright  2023             FORTNA Europe BV                                        |
	|  All Rights Reserved         Netherlands                                             |
	|                                                                                      |
	----------------------------------------------------------------------------------------
	Version history:
	Date        | Version   | Author       | Remark
	----------------------------------------------------------------------------------------
	05/07/2023  | 1.0       | S. Nikodem   | Release TIA 17 | DHL Munich 2023
	13/03/2023  | 1.1       | S. Nieswiec  | Updated for new Baseline
	02/05/2024  | 1.2       | J.Majer      | Datatype conversions changed from automatic to explicit, to accomodate IEC 61131-3 standard

	*)

	REGION New data recived

	    IF NOT (#iq_UDT_MFCParcelDestination.ObjectID <> '')
	        AND NOT (#iq_UDT_MFCParcelDestination.ObjectID <> '0000000000')
	        AND NOT (#iq_UDT_MFCParcelDestination.ObjectID <> '0')
	    THEN

	        //Counter only for statistics
	        #ss_Counter.NewData += 1;

	        //Reset GIN number
	        #sx_NewDataGinNumber := 0;

	        //Find the Object ID in DB_GIN
	        FOR #ti_GINLoop := #ii_GINRangeStart TO #ii_GINRangeEnd DO

	            IF "DB_GIN".GIN[#ti_GINLoop].DHL.ObjectID = #iq_UDT_MFCParcelDestination.ObjectID THEN

	                //Save GIN number
	                #sx_NewDataGinNumber := #ti_GINLoop;

	                //Copy data to DB_GIN
	                "DB_GIN".GIN[#sx_NewDataGinNumber].DHL.SortStrategy := #iq_UDT_MFCParcelDestination.SortStrategy;
	                "DB_GIN".GIN[#sx_NewDataGinNumber].DHL.Destination[1].ID := #iq_UDT_MFCParcelDestination.Destination_1;
	                "DB_GIN".GIN[#sx_NewDataGinNumber].DHL.Destination[2].ID := #iq_UDT_MFCParcelDestination.Destination_2;
	                "DB_GIN".GIN[#sx_NewDataGinNumber].DHL.Destination[3].ID := #iq_UDT_MFCParcelDestination.Destination_3;
	                "DB_GIN".GIN[#sx_NewDataGinNumber].DHL.Destination[4].ID := #iq_UDT_MFCParcelDestination.Destination_4;
	                "DB_GIN".GIN[#sx_NewDataGinNumber].DHL.Destination[5].ID := #iq_UDT_MFCParcelDestination.Destination_5;
	                "DB_GIN".GIN[#sx_NewDataGinNumber].DHL.Destination[6].ID := #iq_UDT_MFCParcelDestination.Destination_6;

	                //Check if destination message is resent
	                IF "DB_GIN".GIN[#sx_NewDataGinNumber].DHL.MFCMessage.Received.Destination THEN

	                    "DB_GIN".GIN[#sx_NewDataGinNumber].DHL.MFCMessage.Received.DestinationResent := True;

	                    //Counter only for statistics
	                    #ss_Counter.DestinationResent += 1;

	                    //Check whether the parcel can be delivered to the new destination.
	                    //Destination 0-5
	                    FOR #ti_DestinationLoop := 0 TO 5 DO

	                        IF (("DB_GIN".GIN[#sx_NewDataGinNumber].General.Destination[#ti_DestinationLoop] > "DB_GIN".GIN[1].DHL.ParcelLocation.Current) AND NOT ("DB_GIN".GIN[1].DHL.ParcelLocation.Current = 0))
	                            OR (("DB_GIN".GIN[#sx_NewDataGinNumber].General.Destination[#ti_DestinationLoop] > "DB_GIN".GIN[1].DHL.ParcelLocation.Last) AND NOT ("DB_GIN".GIN[1].DHL.ParcelLocation.Last = 0))
	                        THEN

	                            #FB_MFC_Sort_SortResult_Instance(is_ObjectID := "DB_GIN".GIN[#ti_GINLoop].DHL.ObjectID,
	                                                             ii_DischargeLocation := DINT_TO_UINT("DB_GIN".GIN[#sx_NewDataGinNumber].General.Destination[#ti_DestinationLoop]),
	                                                             ii_Result := 2,
	                                                             ii_Reason := 5,
	                                                             ii_SourceNode := #ii_SourceNode,
	                                                             ii_DestinationNode := #ii_DestinationNode,
	                                                             iq_UDT_FifoHeader := #iq_UDT_FifoHeader,
	                                                             iqs_FifoData := #iqs_FifoData,
	                                                             iqdi_MessageSequenceNumber := #iqdi_MessageSequenceNumber);

	                            //Counter only for statistics
	                            #ss_Counter.LateDestination += 1;

	                        END_IF;

	                    END_FOR;

	                END_IF;

	                //Destination message received
	                "DB_GIN".GIN[#sx_NewDataGinNumber].DHL.MFCMessage.Received.Destination := True;

	                //Counter only for statistics
	                #ss_Counter.CombinedData += 1;

	                EXIT;

	            END_IF;

	        END_FOR;

	        //Check if GIN number match with Object ID
	        IF #sx_NewDataGinNumber = 0 THEN

	            //Counter only for statistics
	            #ss_Counter.DataNotMerged += 1;

	        END_IF;

	        //Reset structure
	        #iq_UDT_MFCParcelDestination.ObjectID := '';
	        #iq_UDT_MFCParcelDestination.SortStrategy := '';
	        #iq_UDT_MFCParcelDestination.Destination_1 := 0;
	        #iq_UDT_MFCParcelDestination.Destination_2 := 0;
	        #iq_UDT_MFCParcelDestination.Destination_3 := 0;
	        #iq_UDT_MFCParcelDestination.Destination_4 := 0;
	        #iq_UDT_MFCParcelDestination.Destination_5 := 0;
	        #iq_UDT_MFCParcelDestination.Destination_6 := 0;

	    END_IF;

	END_REGION

END_FUNCTION_BLOCK

FUNCTION_BLOCK "FB_MFC_Sort_Heartbeat"
{ S7_Optimized_Access := 'TRUE' }
VERSION : 0.1
// ATTRIBUTES
// AUTO_NUMBER = True
// BLOCK_NUMBER = 120
// END_ATTRIBUTES
   VAR_INPUT
      iudi_HeartbeatInterval { ExternalAccessible := 'False'; ExternalVisible := 'False'; ExternalWritable := 'False'} : UDInt;   // Heartbeat send time interval [ms]
      ii_SourceNode { ExternalAccessible := 'False'; ExternalVisible := 'False'; ExternalWritable := 'False'} : Int;   // ID Source Node
      ii_DestinationNode { ExternalAccessible := 'False'; ExternalVisible := 'False'; ExternalWritable := 'False'} : Int;   // ID Destination Node
   END_VAR

   VAR_OUTPUT
      qx_Error { ExternalAccessible := 'False'; ExternalVisible := 'False'; ExternalWritable := 'False'} : Bool;   // TRUE when collective block error occurred
      qx_Warning { ExternalAccessible := 'False'; ExternalVisible := 'False'; ExternalWritable := 'False'} : Bool;   // TRUE when collective block warning occurred
   END_VAR

   VAR_IN_OUT
      iq_UDT_FifoHeader : "UDT_FifoHeader";   // FIFO header
      iqs_FifoData : Array[*] of "UDT_MessageV2";   // FIFO data buffer
      iqdi_MessageSequenceNumber { ExternalAccessible := 'False'; ExternalVisible := 'False'; ExternalWritable := 'False'} : Int;   // Message number
   END_VAR

   VAR
      ss_FB_HeartbeatPulse { ExternalAccessible := 'False'; ExternalVisible := 'False'; ExternalWritable := 'False'; S7_SetPoint := 'False'} : "FB_Pulse";   // Heartbeat send pulse generator
      s_UDT_MessageArray { ExternalAccessible := 'False'; ExternalVisible := 'False'; ExternalWritable := 'False'; S7_SetPoint := 'False'} : "UDT_MessageV2";   // Message array byte
      s_UDT_MessageHeader { ExternalAccessible := 'False'; ExternalVisible := 'False'; ExternalWritable := 'False'; S7_SetPoint := 'False'} : "UDT_MFCSortMessageHeader";   // Message header
      ss_MessageBody { ExternalAccessible := 'False'; ExternalVisible := 'False'; ExternalWritable := 'False'} : Struct   // Message body
         MsgID { ExternalAccessible := 'False'; ExternalVisible := 'False'; ExternalWritable := 'False'} : Word;   // Message ID
         MsgLength { ExternalAccessible := 'False'; ExternalVisible := 'False'; ExternalWritable := 'False'} : Word;   // Message length
         Eom { ExternalAccessible := 'False'; ExternalVisible := 'False'; ExternalWritable := 'False'} : Byte;   // End of message
      END_STRUCT;
      ss_Status { ExternalAccessible := 'False'; ExternalVisible := 'False'; ExternalWritable := 'False'} : Struct   // Status structure
         FIFOStatus { ExternalAccessible := 'False'; ExternalVisible := 'False'; ExternalWritable := 'False'} : "UDT_FifoStatus";
         FIFOError { ExternalAccessible := 'False'; ExternalVisible := 'False'; ExternalWritable := 'False'; S7_SetPoint := 'True'} : Bool;   //  FIFO error
         FIFOWarning { ExternalAccessible := 'False'; ExternalVisible := 'False'; ExternalWritable := 'False'; S7_SetPoint := 'True'} : Bool;   // FIFO warning
         InvalidMessageArraySize { ExternalAccessible := 'False'; ExternalVisible := 'False'; ExternalWritable := 'False'} : Bool;   // Message array is too short for message
         InvalidTimeInterval { ExternalAccessible := 'False'; ExternalVisible := 'False'; ExternalWritable := 'False'} : Bool;   // Heartbeat time interval lower than zero
      END_STRUCT;
      sdi_SerializePosition { ExternalAccessible := 'False'; ExternalVisible := 'False'; ExternalWritable := 'False'} : DInt;   // Position in array where serialize finished writing data +1
      si_MaximumMessageLength { ExternalAccessible := 'False'; ExternalVisible := 'False'; ExternalWritable := 'False'} : Int;   // Maximum number of elements in message array
      si_SerializeStatus { ExternalAccessible := 'False'; ExternalVisible := 'False'; ExternalWritable := 'False'} : Int;   // Function serialize status
      sx_HeartbeatPulse { ExternalAccessible := 'False'; ExternalVisible := 'False'; ExternalWritable := 'False'} : Bool;   // Heartbeat pulse
   END_VAR

   VAR CONSTANT
      ci_MessageLength : Word := 16#0004;   // 10#0004 = 16#0004 - Message length
      ci_Som : Byte := 16#FD;   // Start of message
      ci_Eom : Byte := 16#FE;   // End of message
      ci_MsgID : Word := 16#005A;   // 10#0090 = 16#005A - Message ID
      ci_MsgLength : Word := 16#0000;   // 10#0000 = 16#0000 - Message length
   END_VAR


BEGIN
	(*
	----------------------------------------------------------------------------------------
	|                                                                                      |
	|  Copyright  2023             FORTNA Europe BV                                        |
	|  All Rights Reserved         Netherlands                                             |
	|                                                                                      |
	----------------------------------------------------------------------------------------
	Version history:
	Date        | Version   | Author       | Remark
	----------------------------------------------------------------------------------------
	05/01/2023  | 1.0       | S. Nikodem   | Release TIA 17 | DHL Munich 2023
	13/03/2023  | 1.1       | S. Nieswiec  | Updated for new Baseline
	02/05/2024  | 1.2       | J.Majer      | Datatype conversions changed from automatic to explicit, to accomodate IEC 61131-3 standard

	*)

	REGION 1 – FIFO header status update

	    // Mode 'S' - FIFO register status update.
	    "FC_Fifo"(ic_Mode := 'S',
	              qUDT_Status => #ss_Status.FIFOStatus,
	              qx_Error => #ss_Status.FIFOError,
	              qx_Warning => #ss_Status.FIFOWarning,
	              iqv_Data := #s_UDT_MessageArray,
	              iqUDT_FifoHeader := #iq_UDT_FifoHeader,
	              iqv_DataBuffer := #iqs_FifoData);

	END_REGION

	REGION 2 – Heartbeat interval validation

	    // Check Heartbeat interval.
	    #ss_Status.InvalidTimeInterval := #iudi_HeartbeatInterval <= 0;

	END_REGION

	REGION 3 – Message array size validation

	    // Get size of the array.
	    #si_MaximumMessageLength := "FC_GetNrOfArrayEl"(#s_UDT_MessageArray.Bytes);

	    // Message array size validation.
	    #ss_Status.InvalidMessageArraySize := WORD_TO_INT(#ci_MessageLength) > #si_MaximumMessageLength;

	END_REGION

	REGION 4 – Generate heartbeat pulse

	    IF NOT #ss_Status.InvalidTimeInterval
	        AND NOT #ss_Status.InvalidMessageArraySize
	    THEN
	        // Heartbeat pulse generator.
	        #ss_FB_HeartbeatPulse(iudi_PulseTime := #iudi_HeartbeatInterval,
	                              qx_Pulse => #sx_HeartbeatPulse);
	    END_IF;

	END_REGION

	REGION 5 – Message preparation

	    // FIFO full check.
	    IF NOT #iq_UDT_FifoHeader.Status.Full
	    THEN
	        // Errors and send pulse check.
	        IF NOT #ss_Status.FIFOError
	            AND NOT #ss_Status.InvalidMessageArraySize
	            AND #sx_HeartbeatPulse
	        THEN

	            REGION 5.1 – Header preparation

	                // Check sequence number. If it is equal or greater than 255 reset it to 1.
	                IF #iqdi_MessageSequenceNumber <= 255
	                THEN
	                    #iqdi_MessageSequenceNumber += 1;
	                ELSE
	                    #iqdi_MessageSequenceNumber := 1;
	                END_IF;

	                // Write parts of the header into structure.
	                #s_UDT_MessageHeader.SOM := #ci_Som;
	                #s_UDT_MessageHeader.SourceNode := INT_TO_BYTE(#ii_SourceNode);
	                #s_UDT_MessageHeader.DestinationNode := INT_TO_BYTE(#ii_DestinationNode);
	                #s_UDT_MessageHeader.SeqNumber := INT_TO_BYTE(#iqdi_MessageSequenceNumber);
	                #s_UDT_MessageHeader.DataLength := #ci_MessageLength;
	                #s_UDT_MessageHeader.NumMsg := 1;

	                #ss_MessageBody.MsgID := #ci_MsgID;
	                #ss_MessageBody.MsgLength := #ci_MsgLength;
	                #ss_MessageBody.Eom := #ci_Eom;

	            END_REGION

	            REGION 5.2 – Convert message into array of bytes

	                // Initialize the header serialize position and convert header structure into array of bytes.
	                #sdi_SerializePosition := 0;
	                #si_SerializeStatus := Serialize(SRC_VARIABLE := #s_UDT_MessageHeader,
	                                                 DEST_ARRAY => #s_UDT_MessageArray.Bytes,
	                                                 POS := #sdi_SerializePosition);

	                // Initialize the body serialize position and convert header structure into array of bytes
	                #si_SerializeStatus := Serialize(SRC_VARIABLE := #ss_MessageBody,
	                                                 DEST_ARRAY => #s_UDT_MessageArray.Bytes,
	                                                 POS := #sdi_SerializePosition);

	            END_REGION

	            REGION 5.3 – Write message into the FIFO buffer

	                // Mode 'W' - Write FIFO record.
	                "FC_Fifo"(ic_Mode := 'W',
	                          qUDT_Status => #ss_Status.FIFOStatus,
	                          qx_Error => #ss_Status.FIFOError,
	                          qx_Warning => #ss_Status.FIFOWarning,
	                          iqv_Data := #s_UDT_MessageArray,
	                          iqUDT_FifoHeader := #iq_UDT_FifoHeader,
	                          iqv_DataBuffer := #iqs_FifoData);

	            END_REGION

	        END_IF;
	    ELSE
	        // If FIFO is full set FIFO main and FIFO full errors.
	        #ss_Status.FIFOError := TRUE;
	        #ss_Status.FIFOStatus.FifoFull := TRUE;
	    END_IF;

	END_REGION

	REGION 6 - Status

	    // Parametrization collective error output.
	    #qx_Error :=
	    #ss_Status.FIFOError
	    OR #ss_Status.InvalidTimeInterval
	    OR #ss_Status.InvalidMessageArraySize;

	    // Parametrization collective warning output.
	    #qx_Warning := #ss_Status.FIFOWarning;

	END_REGION
END_FUNCTION_BLOCK

FUNCTION_BLOCK "FB_MFC_Sort_COY_Decode"
{ S7_Optimized_Access := 'TRUE' }
VERSION : 1.1
// ATTRIBUTES
// AUTO_NUMBER = True
// BLOCK_NUMBER = 114
// END_ATTRIBUTES
   VAR_INPUT
      iudi_HeartbeatTimeout { ExternalAccessible := 'False'; ExternalVisible := 'False'; ExternalWritable := 'False'} : UDInt;   // Heartbeat timeout [ms]
      ix_Connected { ExternalAccessible := 'False'; ExternalVisible := 'False'; ExternalWritable := 'False'} : Bool;   // TRUE when HB monitoring enable
      ix_ResetData { ExternalAccessible := 'False'; ExternalVisible := 'False'; ExternalWritable := 'False'} : Bool;   // TRUE when reset statistics required
   END_VAR

   VAR_OUTPUT
      qx_Error { ExternalAccessible := 'False'; ExternalVisible := 'False'; ExternalWritable := 'False'} : Bool;   // TRUE when collective block error occurred
      qx_Warning { ExternalAccessible := 'False'; ExternalVisible := 'False'; ExternalWritable := 'False'} : Bool;   // TRUE when collective block warningoccurred
   END_VAR

   VAR_IN_OUT
      iq_UDT_Statistics : "UDT_DecodeStatistics";   // Decode statistics
      iq_UDT_FifoReceiveHeader : "UDT_FifoHeader";   // FIFO receive header
      iqa_FifoReceiveData : Array[*] of "UDT_MessageV2";   // FIFO receive data
      iq_UDT_MessageData : "UDT_MFCSortCOYMessageData";   // Received message data
      iqx_Reconnect { ExternalAccessible := 'False'; ExternalVisible := 'False'; ExternalWritable := 'False'} : Bool;   // Reconnect connection
   END_VAR

   VAR
      s_FB_TimerHeartbeatCheck { ExternalAccessible := 'False'; ExternalVisible := 'False'; ExternalWritable := 'False'; S7_SetPoint := 'False'} : "FB_TimerOnOffDelay";   // "FB_TimerOnOffDelay" - to measure the time of missing HB
      s_UDT_FifoMessage { ExternalAccessible := 'False'; ExternalVisible := 'False'; ExternalWritable := 'False'; S7_SetPoint := 'False'} : "UDT_MessageV2";   // Buffer for fifos message
      s_R_TRIG_Connected {InstructionName := 'R_TRIG'; LibVersion := '1.0'; ExternalAccessible := 'False'; ExternalVisible := 'False'; ExternalWritable := 'False'; S7_SetPoint := 'False'} : R_TRIG;   // Siemens "R_TRIG" - to prepare the rising edge trigger on "ix_Connected" signal
      s_F_TRIG_HeartbeatNotOk {InstructionName := 'F_TRIG'; LibVersion := '1.0'; ExternalAccessible := 'False'; ExternalVisible := 'False'; ExternalWritable := 'False'; S7_SetPoint := 'False'} : F_TRIG;   // Siemens "F_TRIG" - to prepare the falling edge trigger on "sx_HeartbeatOk" signal
      ss_CounterRecivedMessage { ExternalAccessible := 'False'; ExternalVisible := 'False'; ExternalWritable := 'False'} : Struct   // Counters with recived messages
         Heartbeat { ExternalAccessible := 'False'; ExternalVisible := 'False'; ExternalWritable := 'False'} : UDInt;   // "Heartbeat" message
         MFCEvent { ExternalAccessible := 'False'; ExternalVisible := 'False'; ExternalWritable := 'False'} : UDInt;   // "MFCEvent" message
         SystemStatusRequest { ExternalAccessible := 'False'; ExternalVisible := 'False'; ExternalWritable := 'False'} : UDInt;   // "SystemStatusRequest" message
         SetSystemMode { ExternalAccessible := 'False'; ExternalVisible := 'False'; ExternalWritable := 'False'} : UDInt;   // "SetSystemMode" message
         SetSystemStatus { ExternalAccessible := 'False'; ExternalVisible := 'False'; ExternalWritable := 'False'} : UDInt;   // "SetSystemStatus" message
         XrayRegistrationInfo { ExternalAccessible := 'False'; ExternalVisible := 'False'; ExternalWritable := 'False'} : UDInt;   // "XrayRegistrationInfo" message
         InvalidMessageID { ExternalAccessible := 'False'; ExternalVisible := 'False'; ExternalWritable := 'False'} : UDInt;   // "InvalidMessageID" message
      END_STRUCT;
      ss_CounterInvalidDestination { ExternalAccessible := 'False'; ExternalVisible := 'False'; ExternalWritable := 'False'} : Struct   // Counters with invalid destination ranges
         Destination_1 { ExternalAccessible := 'False'; ExternalVisible := 'False'; ExternalWritable := 'False'} : UDInt;
         Destination_2 { ExternalAccessible := 'False'; ExternalVisible := 'False'; ExternalWritable := 'False'} : UDInt;
         Destination_3 { ExternalAccessible := 'False'; ExternalVisible := 'False'; ExternalWritable := 'False'} : UDInt;
         Destination_4 { ExternalAccessible := 'False'; ExternalVisible := 'False'; ExternalWritable := 'False'} : UDInt;
         Destination_5 { ExternalAccessible := 'False'; ExternalVisible := 'False'; ExternalWritable := 'False'} : UDInt;
         Destination_6 { ExternalAccessible := 'False'; ExternalVisible := 'False'; ExternalWritable := 'False'} : UDInt;
      END_STRUCT;
      ss_Status { ExternalAccessible := 'False'; ExternalVisible := 'False'; ExternalWritable := 'False'} : Struct   // Status structure
         BadMessage { ExternalAccessible := 'False'; ExternalVisible := 'False'; ExternalWritable := 'False'} : Array[1..10] of "UDT_BytesMessage";   //     Unknown message read
         FIFOReceiveStatus { ExternalAccessible := 'False'; ExternalVisible := 'False'; ExternalWritable := 'False'} : "UDT_FifoStatus";   //     Receive FIFO status structure
         FIFOReceiveError { ExternalAccessible := 'False'; ExternalVisible := 'False'; ExternalWritable := 'False'; S7_SetPoint := 'True'} : Bool;   //     FIFO error
         FIFOReceiveWarning { ExternalAccessible := 'False'; ExternalVisible := 'False'; ExternalWritable := 'False'} : Bool;   //     FIFO warning
         InvalidTimeout { ExternalAccessible := 'False'; ExternalVisible := 'False'; ExternalWritable := 'False'} : Bool;   //     Invalid Heartbeat timeout
      END_STRUCT;
      ss_MessageStructure { ExternalAccessible := 'False'; ExternalVisible := 'False'; ExternalWritable := 'False'} : Struct   // Received a message structure
         PieceID { ExternalAccessible := 'False'; ExternalVisible := 'False'; ExternalWritable := 'False'} : String[16];   // Piece ID
         VID { ExternalAccessible := 'False'; ExternalVisible := 'False'; ExternalWritable := 'False'} : String[40];   // VID
         RoutingCode { ExternalAccessible := 'False'; ExternalVisible := 'False'; ExternalWritable := 'False'} : String[1];   // RoutingCode
      END_STRUCT;
      sdi_SerializePosition { ExternalAccessible := 'False'; ExternalVisible := 'False'; ExternalWritable := 'False'} : DInt;   // Position in array where serialize finished writing data +1
      si_SerializeStatus { ExternalAccessible := 'False'; ExternalVisible := 'False'; ExternalWritable := 'False'} : Int;   // Function serialize status
      si_MessageID { ExternalAccessible := 'False'; ExternalVisible := 'False'; ExternalWritable := 'False'} : Int;   // Message ID
      si_RingBufferNumber { ExternalAccessible := 'False'; ExternalVisible := 'False'; ExternalWritable := 'False'} : Int := 1;   // Bad messages ringbuffer counter
      si_LocationIdentifier { ExternalAccessible := 'False'; ExternalVisible := 'False'; ExternalWritable := 'False'} : UInt;   // Location identifier
      sx_Heartbeat { ExternalAccessible := 'False'; ExternalVisible := 'False'; ExternalWritable := 'False'} : Bool;   // Heartbeat message detected
      sx_HeartbeatOK { ExternalAccessible := 'False'; ExternalVisible := 'False'; ExternalWritable := 'False'} : Bool;   // Heartbeat ok
   END_VAR

   VAR_TEMP
      ta_MessageData : Array[0..3] of Byte;   // Messages ID
      ta_MessageData_1 : Array[0..1] of Byte;   // Messages ID
      tdi_NumericValue : UDInt;   // Numeric Value
      ti_BadMessageSize : Int;   // Bad message buffer size
      ti_NumberOfMessageBytes : Int;   // Length of FIFO message
      ti_NumericValue : Int;   // Numeric Value
      ti_Loop : Int;   // Loop counter
      ti_SystemStatus : Int;
      ti_NrOfArrayElements : Int;   // Number of array elements
      tx_MessageRead : Bool;   // Message read from FIFO
      tx_InvalidHeader : Bool;   // Invalid header
      tx_InvalidMessageID : Bool;   // Invalid message ID
      tx_BadMessage : Bool;   // Message with prohibited data
      ts_RoutingCode : String;
   END_VAR

   VAR CONSTANT
      ci_DestinationMin : Int := 351;   // Minimum value of the destination
      ci_DestinationMax : Int := 355;   // Maximum value of the destination
   END_VAR


BEGIN
	(*
	----------------------------------------------------------------------------------------
	|                                                                                      |
	|  Copyright  2023             FORTNA Europe BV                                        |
	|  All Rights Reserved         Netherlands                                             |
	|                                                                                      |
	----------------------------------------------------------------------------------------
	Version history:
	Date        | Version   | Author       | Remark
	----------------------------------------------------------------------------------------
	15/02/2023  | 1.0       | S. Nikodem   | Release TIA 17 | DHL Munich 2023
	23/08/2023  | 1.1       | S.Theccharis | bug fix on bit pattern
	12/09/2023  | 1.2       | S. Nikodem   | Dynamic array length detection
	06/02/2023  | 1.3       | M.Diebel     | Read array from 0 position
	13/03/2023  | 1.4       | S. Nieswiec  | Updated for new Baseline
	*)

	REGION 1 – FIFO header status update

	    // Mode 'S' - FIFO register status update.
	    "FC_Fifo"(ic_Mode := 'S',
	              qUDT_Status => #ss_Status.FIFOReceiveStatus,
	              qx_Error => #ss_Status.FIFOReceiveError,
	              qx_Warning => #ss_Status.FIFOReceiveWarning,
	              iqv_Data := #s_UDT_FifoMessage,
	              iqUDT_FifoHeader := #iq_UDT_FifoReceiveHeader,
	              iqv_DataBuffer := #iqa_FifoReceiveData);

	    // FIFO isn't empty and doesn't have error.
	    IF NOT #iq_UDT_FifoReceiveHeader.Status.Empty
	        AND NOT #ss_Status.FIFOReceiveError
	    THEN
	        // Mode 'R' - Read FIFO record.
	        "FC_Fifo"(ic_Mode := 'R',
	                  qUDT_Status => #ss_Status.FIFOReceiveStatus,
	                  qx_Error => #ss_Status.FIFOReceiveError,
	                  qx_Warning => #ss_Status.FIFOReceiveWarning,
	                  iqv_Data := #s_UDT_FifoMessage,
	                  iqUDT_FifoHeader := #iq_UDT_FifoReceiveHeader,
	                  iqv_DataBuffer := #iqa_FifoReceiveData);

	        // Message read bit set.
	        #tx_MessageRead := TRUE;

	        // FIFO empty or FIFO error occured.
	    ELSE
	        #tx_MessageRead := FALSE;
	    END_IF;

	END_REGION

	REGION 2 – Message type recognition

	    IF #tx_MessageRead
	    THEN

	        #ta_MessageData[0] := #s_UDT_FifoMessage.Bytes[0];
	        #ta_MessageData[1] := #s_UDT_FifoMessage.Bytes[1];

	        // Deserialize Message ID
	        #sdi_SerializePosition := 0;
	        #si_SerializeStatus := Deserialize(SRC_ARRAY := #ta_MessageData,
	                                           DEST_VARIABLE => #si_MessageID,
	                                           POS := #sdi_SerializePosition);

	        CASE #si_MessageID OF
	            90:  //Heartbeat
	                #sx_Heartbeat := TRUE;

	                //Only statistics
	                #ss_CounterRecivedMessage.Heartbeat += 1;

	            104:  //MFC Event

	                //Get the number of event from the reviced message
	                #ta_MessageData_1[0] := #s_UDT_FifoMessage.Bytes[4];
	                #ta_MessageData_1[1] := #s_UDT_FifoMessage.Bytes[5];

	                #sdi_SerializePosition := 0;
	                #si_SerializeStatus := Deserialize(SRC_ARRAY := #ta_MessageData,
	                                                   DEST_VARIABLE => #iq_UDT_MessageData.MFCEvent.Event,
	                                                   POS := #sdi_SerializePosition);

	                #iq_UDT_MessageData.MFCEvent.Action := BYTE_TO_INT(#s_UDT_FifoMessage.Bytes[6]);
	                #iq_UDT_MessageData.MFCEvent.Settings := BYTE_TO_INT(#s_UDT_FifoMessage.Bytes[7]);

	                //Only statistics
	                #ss_CounterRecivedMessage.MFCEvent += 1;

	            105:  //System status request

	                #iq_UDT_MessageData.SystemStatusRequest.UpdateStatus := TRUE;

	                //Only statistics
	                #ss_CounterRecivedMessage.SystemStatusRequest += 1;

	            106:  //Set system mode

	                //Get location identifier from the reviced message
	                #ta_MessageData_1[0] := #s_UDT_FifoMessage.Bytes[4];
	                #ta_MessageData_1[1] := #s_UDT_FifoMessage.Bytes[5];

	                #sdi_SerializePosition := 0;
	                #si_SerializeStatus := Deserialize(SRC_ARRAY := #ta_MessageData_1,
	                                                   DEST_VARIABLE => #si_LocationIdentifier,
	                                                   POS := #sdi_SerializePosition);

	                #ti_NrOfArrayElements := "FC_GetNrOfArrayEl"(#iq_UDT_MessageData.System);

	                //Matching identifier
	                FOR #ti_Loop := 0 TO (#ti_NrOfArrayElements - 1) DO

	                    IF #si_LocationIdentifier = #iq_UDT_MessageData.System[#ti_Loop].LocationIdentifier THEN

	                        //System mode - bit value

	                        //Get location identifier from the reviced message
	                        #ta_MessageData_1[0] := #s_UDT_FifoMessage.Bytes[6];
	                        #ta_MessageData_1[1] := #s_UDT_FifoMessage.Bytes[7];

	                        #sdi_SerializePosition := 0;
	                        #si_SerializeStatus := Deserialize(SRC_ARRAY := #ta_MessageData_1,
	                                                           DEST_VARIABLE => #iq_UDT_MessageData.System[#ti_Loop].Command.Mode,
	                                                           POS := #sdi_SerializePosition);

	                        //System mode - Infeed = 1/Outfeed = 2 - number
	                        IF #iq_UDT_MessageData.System[#ti_Loop].Command.Mode.%X1 THEN

	                            #iq_UDT_MessageData.System[#ti_Loop].Command.SystemMode := 1;

	                        ELSIF #iq_UDT_MessageData.System[#ti_Loop].Command.Mode.%X2 THEN

	                            #iq_UDT_MessageData.System[#ti_Loop].Command.SystemMode := 2;

	                        END_IF;


	                        //System mode - bool value
	                        //Infeed mode
	                        IF #iq_UDT_MessageData.System[#ti_Loop].Command.Mode.%X1 THEN
	                            #iq_UDT_MessageData.System[#ti_Loop].Command.Infeed := True;
	                        ELSE
	                            #iq_UDT_MessageData.System[#ti_Loop].Command.Infeed := False;
	                        END_IF;

	                        //Outfeed mode
	                        IF #iq_UDT_MessageData.System[#ti_Loop].Command.Mode.%X2 THEN
	                            #iq_UDT_MessageData.System[#ti_Loop].Command.Outfeed := True;
	                        ELSE
	                            #iq_UDT_MessageData.System[#ti_Loop].Command.Outfeed := False;
	                        END_IF;

	                        //Contingency mode
	                        IF #iq_UDT_MessageData.System[#ti_Loop].Command.Mode.%X3 THEN
	                            #iq_UDT_MessageData.System[#ti_Loop].Command.Contingency := True;
	                        ELSE
	                            #iq_UDT_MessageData.System[#ti_Loop].Command.Contingency := False;
	                        END_IF;

	                        //Normal operation mode
	                        IF #iq_UDT_MessageData.System[#ti_Loop].Command.Mode.%X4 THEN
	                            #iq_UDT_MessageData.System[#ti_Loop].Command.NormalOperation := True;
	                        ELSE
	                            #iq_UDT_MessageData.System[#ti_Loop].Command.NormalOperation := False;
	                        END_IF;

	                        //Xray screening mode
	                        IF #iq_UDT_MessageData.System[#ti_Loop].Command.Mode.%X5 THEN
	                            #iq_UDT_MessageData.System[#ti_Loop].Command.XrayScreening := True;
	                        ELSE
	                            #iq_UDT_MessageData.System[#ti_Loop].Command.XrayScreening := False;
	                        END_IF;

	                        //Xray transport mode
	                        IF #iq_UDT_MessageData.System[#ti_Loop].Command.Mode.%X6 THEN
	                            #iq_UDT_MessageData.System[#ti_Loop].Command.XrayTransport := True;
	                        ELSE
	                            #iq_UDT_MessageData.System[#ti_Loop].Command.XrayTransport := False;
	                        END_IF;

	                        //Truck line empty mode
	                        IF #iq_UDT_MessageData.System[#ti_Loop].Command.Mode.%X7 THEN
	                            #iq_UDT_MessageData.System[#ti_Loop].Command.TruckLineEmpty := True;
	                        ELSE
	                            #iq_UDT_MessageData.System[#ti_Loop].Command.TruckLineEmpty := False;
	                        END_IF;

	                        //Truck line normal mode
	                        IF #iq_UDT_MessageData.System[#ti_Loop].Command.Mode.%X8 THEN
	                            #iq_UDT_MessageData.System[#ti_Loop].Command.TruckLineNormal := True;
	                        ELSE
	                            #iq_UDT_MessageData.System[#ti_Loop].Command.TruckLineNormal := False;
	                        END_IF;

	                    END_IF;

	                END_FOR;

	                //Only statistics
	                #ss_CounterRecivedMessage.SetSystemMode += 1;

	            107:  //Set system status

	                //Get location identifier from the reviced message
	                #ta_MessageData_1[0] := #s_UDT_FifoMessage.Bytes[4];
	                #ta_MessageData_1[1] := #s_UDT_FifoMessage.Bytes[5];

	                #sdi_SerializePosition := 0;
	                #si_SerializeStatus := Deserialize(SRC_ARRAY := #ta_MessageData_1,
	                                                   DEST_VARIABLE => #si_LocationIdentifier,
	                                                   POS := #sdi_SerializePosition);

	                #ti_NrOfArrayElements := "FC_GetNrOfArrayEl"(#iq_UDT_MessageData.System);

	                //Matching identifier
	                FOR #ti_Loop := 0 TO (#ti_NrOfArrayElements - 1) DO

	                    IF #si_LocationIdentifier = #iq_UDT_MessageData.System[#ti_Loop].LocationIdentifier THEN

	                        #ti_SystemStatus := BYTE_TO_INT(#s_UDT_FifoMessage.Bytes[6]);

	                        CASE #ti_SystemStatus OF
	                            1:
	                                #iq_UDT_MessageData.System[#ti_Loop].Command.Start := True;
	                            2:
	                                #iq_UDT_MessageData.System[#ti_Loop].Command.Stop := True;
	                            3:
	                                #iq_UDT_MessageData.System[#ti_Loop].Command.Reset := True;
	                        END_CASE;

	                    END_IF;

	                END_FOR;

	                //Only statistics
	                #ss_CounterRecivedMessage.SetSystemStatus += 1;

	            301:  //X-RAY REGISTRATION INFO

	                //Object ID
	                #ta_MessageData[0] := #s_UDT_FifoMessage.Bytes[4];
	                #ta_MessageData[1] := #s_UDT_FifoMessage.Bytes[5];
	                #ta_MessageData[2] := #s_UDT_FifoMessage.Bytes[6];
	                #ta_MessageData[3] := #s_UDT_FifoMessage.Bytes[7];


	                #sdi_SerializePosition := 0;
	                #si_SerializeStatus := Deserialize(SRC_ARRAY := #ta_MessageData,
	                                                   DEST_VARIABLE => #tdi_NumericValue,
	                                                   POS := #sdi_SerializePosition);

	                #iq_UDT_MessageData.XrayRegistrationInfo.ObjectID := DELETE(IN := UDINT_TO_STRING(#tdi_NumericValue), L := 1, P := 1);

